	81:	nMoverToCorrect := nMoverToCorrect +1;
		IF nMoverToCorrect <= g_nMoverCount THEN
			fMoverOrientationRead    := ipMoverApplication[nMoverToCorrect].std.P_ActPosition.c; 
			fMoverOrientationCorrect := fMoverOrientationRead;
			 bDoRotationCorrection := FALSE;
			nStatePreparation := nStatePreparation + 1;	
		ELSE
			bDerterminedMoverOrientation := TRUE;
			nStatePreparation := nStatePreparation + 9;	
		END_IF
		
	82:	IF fMoverOrientationCorrect >= 0 THEN
			IF fMoverOrientationCorrect > 360.0 THEN
				fMoverOrientationCorrect := fMoverOrientationCorrect - 180.0;
				bDoRotationCorrection := TRUE;
			ELSE
				nStatePreparation := nStatePreparation + 1;
			END_IF
		ELSE
			IF fMoverOrientationCorrect < 360.0 THEN
				fMoverOrientationCorrect := fMoverOrientationCorrect + 180.0;
				bDoRotationCorrection := TRUE;
			ELSE
				nStatePreparation := nStatePreparation + 1;
			END_IF
		END_IF			
		
		
	83:	IF bDoRotationCorrection THEN
			
			fPosX := ipMoverApplication[nMoverToCorrect].std.P_ActPosition.x;
			fPosY := ipMoverApplication[nMoverToCorrect].std.P_ActPosition.y;
			fPosC := ipMoverApplication[nMoverToCorrect].std.P_ActPosition.c;
	
			CorrectionPos.SetValuesXYC(fPosX, fPosY, fMoverOrientationCorrect);	
	
			ipMoverApplication[nMoverToCorrect].std.SetMoverPosition('Correction', CorrectionPos);
			
			nStatePreparation := nStatePreparation + 1;	
		ELSE
			nStatePreparation := nStatePreparation - 2;
		END_IF
		
	84:
		IF ipMoverApplication[nMoverToCorrect].std.P_SetMoverPosition.Done THEN
			nStatePreparation := nStatePreparation - 3;
		ELSIF ipMoverApplication[nMoverToCorrect].std.P_SetMoverPosition.Error THEN
			nErrorID := ipMoverApplication[nMoverToCorrect].std.P_SetMoverPosition.ErrorID;
			ipVisuMessage.SetErrorMessage('Rotation-Angle modulo adaption', 'MoverPreparation', nStatePreparation, nErrorID);		
		END_IF
		

	90: nStatePreparation := 500;
	
			
	500: // Done
		nStatePreparation := 0;
		MoverPreparation := TRUE;		
			
		
	END_CASE


	ipVisuMessage.StateUpdate(nStatePreparation, 'MoverPreparation');
END_METHOD

METHOD MoverRecovery : BOOL
VAR_INPUT
	bReset	: BOOL;
END_VAR



VAR_INST

	// Dynamic limitations
	fVeloRec           				: LREAL := 250.0;
	fAccelRec    					: LREAL := 3000.0;
	fJerkRec            			: LREAL := 30000.0;
	
	fVeloTurn           			: LREAL :=  1800.0;
	fAccelTurn    					: LREAL :=   720.0;
	fJerkTurn            			: LREAL := 14400.0;		
	

	idx								: UDINT;	
	nTestCounter					: UDINT;
	nStateMoverRecovery				: INT;	
	bAllMoversDone					: BOOL;
	nForCounter						: UDINT;
	bStillBusy						: BOOL;
	nInitPositionToMoveTo			: UDINT;
	bAllMoversAtInitPosition		: BOOL;
	nInitPositionIndex	  			: UDINT;
	nMoverIndex			  			: UDINT;
	nMoversToInitPositionFound		: UDINT;
	nMoverToJoinTrack				: UDINT;
	nMoverToInitPosition			: UDINT;
	bTryMoveX						: BOOL;
	bTryMoveY						: BOOL;
	nCounterMoverToMove				: INT;	
	
	fInitialMoverPosition			: ARRAY [1..gc_nMaxNumberMovers,1..2] OF LREAL;
	bMoverSortedAlready				: ARRAY [1..gc_nMaxNumberMovers] OF BOOL;
	bMoverSkipInitPosition			: ARRAY [1..gc_nMaxNumberMovers] OF BOOL;
	bMoverToInitPosition			: ARRAY [1..gc_nMaxNumberMovers] OF BOOL;
	bMoverAtInitPosition			: ARRAY [1..gc_nMaxNumberMovers] OF BOOL;
	bMoverBlockedByMove				: ARRAY [1..gc_nMaxNumberMovers] OF BOOL;
	bInitPositionBlockedByMove		: ARRAY [1..gc_nMaxNumberMovers] OF BOOL;	
	bInitialMoverPositionDone		: ARRAY [1..gc_nMaxNumberMovers] OF BOOL;
	nMoverOnTheWayToInitPosition	: ARRAY [1..gc_nMaxNumberMovers] OF UDINT;
	fMoverDistanceToInitialPosition	: ARRAY [1..gc_nMaxNumberMovers] OF LREAL;
	fShortestDistance				: ARRAY [1..gc_nMaxNumberMovers] OF LREAL;
	nClosestMoverToInitPosition		: ARRAY [1..gc_nMaxNumberMovers] OF UDINT;
	nInitPositionMoverTable			: ARRAY [1..gc_nMaxNumberMovers] OF UDINT;
	nMoverRecoveryPosition			: ARRAY [1..gc_nMaxNumberMovers] OF UDINT;
	nJoinTrack						: ARRAY [1..gc_nMaxNumberMovers] OF UDINT;	
	
	fRotationMoverPosition			: ARRAY [1..gc_nMaxNumberMovers,1..2] OF LREAL;
	nMoverToRotationPosition		: UDINT;
	nRotationPositionToMoveTo		: UDINT;
	nMoverBackToInitPosition		: UDINT;

	sInfoText						: STRING;
	targetPos            	 		: PositionXYC;
    currentPos			     		: PositionXYC;
	nCmdReturnError					: UDINT;
	
	
//-----------------first Track run

	fTrackLengthTrack1  	: LREAL;
	fTrackLengthTrack2  	: LREAL;	
	fTrackLengthTrack3  	: LREAL;	
	
	bInitRunFlag			: BOOL;
	bInitRunDone			: BOOL;
	bOneMoverMoving			: BOOL;
	bAllMoversStandingStill	: BOOL;
	bMoversQueuing			: BOOL;
	
	TimerWaitForMovement	: TON;	
	
	
	nState 					: INT;	
	nStateInit				: INT;
	
	
	fbInitList				: FB_List;

	fPositionOnTrack			: LREAL;
	nStationIndex				: UINT;
	nNextStationTrackIndex 		: UINT;
	fNextStationWaitingPosition	: LREAL;
	nTrackIndex					: UDINT;
	nNextStationIndex			: UDINT;
	nListIdentifier				: UDINT;
	bFirstMoverIn				: BOOL;
	ClearTrig					: R_TRIG;
	fMoverPosition				: LREAL;
	fMoverVelocity				: LREAL;
	fMoverAcceleration			: LREAL;
	fMoverJerk					: LREAL;
	strInfo						: STRING;
	
	fMoverSpace					: LREAL;
	fWaitingPositionStation01	: LREAL;
	fWaitingPositionStation02	: LREAL;	
	fWaitingPositionStation03	: LREAL;	
	fWaitingPositionStation04	: LREAL;	
	fWaitingPositionStation05b	: LREAL;	
	fWaitingPositionStation05c	: LREAL;
	
	stMoveParameters 	: ST_MoveOnTrackOptions; 
	strInfoHistory		: ARRAY[0..10] OF STRING;
	
	nResult				: DINT;
	sMessage			: STRING;
	
	
	stJoinTrackOptions		: ST_JoinTrackOptions;
	stMoveOptionsCurve		: ST_MoveCOptions;	

	
	
	nMoverToTurnBack				: UDINT;
	fRecoveryRotTarget				: LREAL;
	fRecoveryRotVel					: LREAL :=  360.0;
	fRecoveryRotAcc					: LREAL := 1800.0;
	fRecoveryRotJerk				: LREAL := 9000.0;
	stRotationOptions				: ST_MoveCOptions;
	
	
	LeavOptions	: ST_LeaveTrackOptions;
	
END_VAR


VAR_INST
	nMoverToTurn					: UDINT;

	fbMoverTarget		: FB_MoverTarget;
	nErrorCode			: DINT;
	bError				: BOOL;
	sInfoMessage		: STRING;

	
END_VAR
IF bReset THEN
	nStateMoverRecovery := 0;
	MoverRecovery := TRUE;
END_IF



CASE nStateMoverRecovery OF

	0:	// Starting mover recovery
		nStateMoverRecovery := 50;
			
	(***************************************************************************************)
	(* Mover Recovery Part1: Checking for unfinished rotation                              *)
	(***************************************************************************************)     			
		
	50:		// Turn rotation angle to closets quarter-angle 
			ipVisuMessage.SetInfoMessage('Clearing rotation', 'Recovery', nStateMoverRecovery);

			nMoverToTurn := 0;
			nStateMoverRecovery := nStateMoverRecovery +1;
			
	51:  	nMoverToTurn := nMoverToTurn +1;
			IF nMoverToTurn > g_nMoverCount THEN
				nStateMoverRecovery := nStateMoverRecovery +3;
			ELSE
				IF ipMoverApplication[nMoverToTurn].std.P_IsPresent THEN

					fRecoveryRotTarget 				  := ipMoverApplication[nMoverToTurn].std.P_ClosestQuaterAngle;	
					stRotationOptions.additionalTurns := 0;
					stRotationOptions.direction		  := Tc3_Mc3PlanarMotion.MC_direction.mcDirectionNonModulo;	
					
					ipMoverApplication[nMoverToTurn].std.MoveC('Recovery - unfinished rotation', fRecoveryRotTarget, fRecoveryRotVel, fRecoveryRotAcc, fRecoveryRotAcc, fRecoveryRotJerk, stRotationOptions);
					nStateMoverRecovery := nStateMoverRecovery +1;				
				END_IF	
			END_IF

	52:		IF ipMoverApplication[nMoverToTurn].std.P_MoveC.Done THEN
				nStateMoverRecovery := nStateMoverRecovery -1;	
			ELSIF ipMoverApplication[nMoverToTurn].std.P_MoveC.Error THEN
				nStateMoverRecovery := nStateMoverRecovery +1;	
			END_IF
 
	53:		// Check error ID and react accordingly
			nErrorID := ipMoverApplication[nMoverToTurn].std.P_MoveC.ErrorID;	
			
			// In case rotation is not possible due to collision with another mover proceed without rotation correction.
			IF nErrorID = 33158 THEN
				nStateMoverRecovery := nStateMoverRecovery -2;	
			END_IF
						
	54:		nStateMoverRecovery := 100;		
			
			
	(*******************************************************************************************)
	(* Mover Recovery Part2: Separating all movers and move each of them to a corner position. *)
	(*******************************************************************************************)    			
		
	100: 
		ipVisuMessage.SetInfoMessage('Separating all movers', 'Recovery', nStateMoverRecovery);
		IF fbMoverTarget.Clear() THEN
			nStateMoverRecovery := nStateMoverRecovery +10;
		END_IF
	
	110:
		bError := FALSE;
		FOR idx:=1 TO g_nMoverCount DO
			IF ipMoverApplication[idx].std.P_IsPresent THEN
				fbMoverTarget.AddMover(ipMoverApplication[idx]);
				IF fbMoverTarget.P_ErrorWarningCode < 0 THEN
					bError := TRUE;
				END_IF
			END_IF
		END_FOR
		
		IF bError THEN
			sInfoMessage := fbMoverTarget.P_Info;
		ELSE
			nStateMoverRecovery := nStateMoverRecovery +10;
		END_IF
			
	120:
		fbMoverTarget.AddPosition(120.0, 120.0);
		fbMoverTarget.AddPosition(120.0, 600.0);
		fbMoverTarget.AddPosition(840.0, 600.0);
		fbMoverTarget.AddPosition(840.0, 120.0);
		
		fbMoverTarget.SetDynamics(250.0, 1000.0, 10000.0);
		
		IF fbMoverTarget.P_ErrorWarningCode < 0 THEN
			sInfoMessage := fbMoverTarget.P_Info;
		ELSE
			nStateMoverRecovery := nStateMoverRecovery +10;
		END_IF
		

	130:
		  sMessage := fbMoverTarget.P_Info;
		nErrorCode := fbMoverTarget.P_ErrorWarningCode;	

		IF fbMoverTarget.MoversToTarget() THEN
			nStateMoverRecovery := 300;
		END_IF
					
	
	(***************************************************************************************)
	(* Mover Recovery Part3: All movers join the outer-track							   *)
	(***************************************************************************************)  	
					
			
	300:	// All movers go on track
			ipVisuMessage.SetInfoMessage('All movers join track', 'Recovery', nStateMoverRecovery);
	
			FOR nForCounter := 1 TO g_nMoverCount DO
				IF ipMoverApplication[nForCounter].std.P_SetPosition.x > 480.0 THEN
					nJoinTrack[nForCounter] := 3;	
				ELSE
					nJoinTrack[nForCounter] := 1;	
				END_IF
			END_FOR
			nStateMoverRecovery := nStateMoverRecovery +1;	
				
	301:	IF nMoverToJoinTrack < g_nMoverCount THEN
				nMoverToJoinTrack := nMoverToJoinTrack +1;
				nStateMoverRecovery := nStateMoverRecovery +1;
			ELSE
				nMoverToJoinTrack := 0;
				nStateMoverRecovery := nStateMoverRecovery + 2; 
			END_IF
				
	302:	stJoinTrackOptions.useOrientation := FALSE;
	
			sInfoText := 'Recovery, join TrackID: ';
			sInfoText := CONCAT(sInfoText, UDINT_TO_STRING(nJoinTrack[nMoverToJoinTrack]));
			
			IF ipMoverApplication[nMoverToJoinTrack].std.JoinTrack( sInfoText,
																	ipTrack[nJoinTrack[nMoverToJoinTrack]].std,
																    fVeloRec,
																	fAccelRec,
																	fJerkRec,
																	stJoinTrackOptions )
			THEN
				ipMoverApplication[nMoverToJoinTrack].P_TrackId := nJoinTrack[nMoverToJoinTrack];
				nStateMoverRecovery := nStateMoverRecovery -1;
			END_IF
			
				
			
			
	303:	bDone := TRUE;
			FOR nForCounter := 1 TO g_nMoverCount DO
				bDone := bDone AND ipMoverApplication[nForCounter].std.P_JoinTrack.Done;
			END_FOR
			
			IF bDone THEN
				nStateMoverRecovery := nStateMoverRecovery + 7;
			END_IF
		
	310:  // Wait for all movers on-track
			bDone := TRUE;
			FOR nForCounter := 1 TO g_nMoverCount DO
				bDone := bDone AND ipMoverApplication[nForCounter].std.P_JoinTrack.Done;
			END_FOR
			IF bDone THEN
				nStateMoverRecovery := 400;
			END_IF
	
				
	(***************************************************************************************)
	(* Mover Recovery Part4: Adding all movers to the Initialization-List and sort them    *)
	(*                       ascending.                              				       *)
	(***************************************************************************************)  			
				
	400:	ipVisuMessage.SetInfoMessage('Sorting all movers', 'Recovery', nStateMoverRecovery);
			IF fbInitList.ClearList() THEN
				nStateMoverRecovery := nStateMoverRecovery + 1;
			END_IF
			
	401:	IF fbInitList.ClearTrackOrder() THEN
				nStateMoverRecovery := nStateMoverRecovery + 9;
			END_IF
	
			
	410:	// Adding all movers to the Initialization-List
			FOR nForCounter := 1 TO g_nMoverCount DO
				fbInitList.AddMover(ipMoverApplication[nForCounter].std);
			END_FOR				
			nStateMoverRecovery := nStateMoverRecovery + 10;
			
			
	420: 	// Adding Track-Order to the Initialization-List for Sorting-Order
			IF fbInitList.AddTrack(ipTrack[1].std) > 0 THEN
				nStateMoverRecovery := nStateMoverRecovery + 1;
			ELSE
				 nResult := fbInitList.P_nResult;
				sMessage := fbInitList.P_sMessage;	
			END_IF
			
	421: 	IF fbInitList.AddTrack(ipTrack[3].std) > 0 THEN
				nStateMoverRecovery := nStateMoverRecovery + 1;
			ELSE
				 nResult := fbInitList.P_nResult;
				sMessage := fbInitList.P_sMessage;	
			END_IF			
						
 	422:	nStateMoverRecovery := 450;
				
	450:	// Sorting all movers 
			fbInitList.P_SortingDirection := eSortingDirection.ascending;
			fbInitList.P_SortingOrigin := 0.0;
	
			 nResult := fbInitList.SortList();
			sMessage := fbInitList.P_sMessage;
			
			IF nResult > 0 THEN
				// Sorting succesful - will return the number of movers sorted e.g. 4
				nStateMoverRecovery:= nStateMoverRecovery + 10;
			ELSIF nResult = 0 THEN
				;// Sorting 
			ELSIF nResult < 0 THEN
				// sorting Error - Check error code and error message
				nStateMoverRecovery:= nStateMoverRecovery +1;
			END_IF
			
	451:	// Check error message and act accordingly		
			 nResult := fbInitList.P_nResult;
			sMessage := fbInitList.P_sMessage;				
	
			
	460:	nStateMoverRecovery:= 500;			
	

	
	(***************************************************************************************)
	(* Mover Recovery Part5: Initialization-Run                                            *)
	(*						 - Sending/Adding each mover to its next closest station       *)
	(*						 - From there on each station takes care of the init-run       *)
	(* 						 - Movers will queu in in front of station 01 				   *)
	(***************************************************************************************)  

	500: // Init all variables 
		ipVisuMessage.SetInfoMessage('Mover init-run', 'Recovery', nStateMoverRecovery);
	
					bOneMoverMoving := FALSE;
			bAllMoversStandingStill := FALSE;
					   bInitRunDone := FALSE;
	
				   nStateMoverRecovery := nStateMoverRecovery + 10;
	
	510: // Check for next Mover
		IF fbInitList.P_FirstInList <> 0 THEN
				 nMoverIndex := fbInitList.P_FirstInList.P_Id;
				 nTrackIndex := ipMoverApplication[nMoverIndex].P_TrackId;
			fPositionOnTrack := ipMoverApplication[nMoverIndex].std.P_SetOnTrack.SetPos;
			
			      bFirstMoverIn := TRUE;
			nStateMoverRecovery := nStateMoverRecovery + 10;
		ELSE
			IF bFirstMoverIn THEN
				nStateMoverRecovery := 600;
			ELSE
				// Init-Run completed
				bInitRunFlag := FALSE;
				nStateMoverRecovery := 1000;	
			END_IF
		END_IF
			
		
	520: // Figuring out the next station the mover has to travel to:
		fMoverSpace := 155.0 + 5.0;
	
		fWaitingPositionStation01	:= ipTrack[1].P_TrackLength/2.0 - fMoverSpace;	
		fWaitingPositionStation02	:= ipTrack[2].P_TrackLength/2.0 - fMoverSpace;	
		fWaitingPositionStation03	:= ipTrack[3].P_TrackLength/2.0 - fMoverSpace;
		fWaitingPositionStation04	:= ipTrack[1].P_TrackLength - fMoverSpace;	
		fWaitingPositionStation05b	:= ipTrack[3].P_TrackLength - fMoverSpace;	
		fWaitingPositionStation05c	:= ipTrack[2].P_TrackLength - fMoverSpace;	
	
		nListIdentifier := 0;
		CASE nTrackIndex OF		
		1:	// Mover on Track01 / Station01
			IF fPositionOnTrack <= fWaitingPositionStation01 THEN
				nNextStationIndex := 1;
				  nListIdentifier := 11;
			ELSE
				nNextStationIndex := 4;
				  nListIdentifier := 14;
			END_IF	
	
		2:	// Mover on Track02 / Station02
			IF fPositionOnTrack <= fWaitingPositionStation02 THEN
				nNextStationIndex := 2;
				  nListIdentifier := 22;
			ELSE
				nNextStationIndex := 5;
				  nListIdentifier := 25;
			END_IF			
		
		3:	// Mover on Track03 / Station 03
			IF fPositionOnTrack <= fWaitingPositionStation03 THEN
				nNextStationIndex := 3;
				  nListIdentifier := 33;
			ELSE
				nNextStationIndex := 5;
				  nListIdentifier := 35;
			END_IF			
		END_CASE
		
		nStateMoverRecovery := nStateMoverRecovery + 10;
			
			
	530: // Calculating the position the mover has to move to next:
		nNextStationTrackIndex := 0;
		
		CASE nNextStationIndex OF
			1:	nNextStationTrackIndex      := 1;
				fNextStationWaitingPosition	:= fWaitingPositionStation01;	
			
			2:	nNextStationTrackIndex      := 2;
				fNextStationWaitingPosition	:= fWaitingPositionStation02;			
			
			3:	nNextStationTrackIndex      := 3;
				fNextStationWaitingPosition	:= fWaitingPositionStation01;			
			
			4:	nNextStationTrackIndex      := 1;
				fNextStationWaitingPosition	:= fWaitingPositionStation04;				
				
			5:	IF nTrackIndex = 2 THEN
					nNextStationTrackIndex := 2;
					fNextStationWaitingPosition	:= fWaitingPositionStation05c;	
				ELSIF nTrackIndex = 3 THEN
					nNextStationTrackIndex := 3;
					fNextStationWaitingPosition	:= fWaitingPositionStation05b;	
				END_IF									
		END_CASE
			
		IF nNextStationTrackIndex > 0 THEN
			nStateMoverRecovery := nStateMoverRecovery + 10;
		END_IF
	
	
	540: 	// Send mover to the next station
			fMoverPosition     := fNextStationWaitingPosition;
			fMoverVelocity     :=    300.0;
			fMoverAcceleration :=  1_000.0;
			fMoverJerk         := 10_000.0;	
	
			stMoveParameters.direction := Tc3_Mc3PlanarMotion.MC_DIRECTION.mcDirectionPositive;
			stMoveParameters.gap       := 240.0;
			
			strInfo := 'Recovery: ';
			strInfo := CONCAT(strInfo, ' Mover: ');
			strInfo := CONCAT(strInfo, UDINT_TO_STRING(nMoverIndex));
			strInfo := CONCAT(strInfo, ' move to Station:' );
			strInfo := CONCAT(strInfo, UDINT_TO_STRING(nNextStationIndex));
			
		
			IF NOT ipMoverApplication[nMoverIndex].std.P_MoveOnTrack.Busy THEN
	
				FOR idx:=10 TO 1 BY -1 DO 
					strInfoHistory[idx] := strInfoHistory[idx-1];
				END_FOR
				strInfoHistory[0] := strInfo;		
			
				ipMoverApplication[nMoverIndex].std.MoveOnTrack( strInfo,
																 ipTrack[nNextStationTrackIndex].std,
																 fMoverPosition,
																 fMoverVelocity,
																 fMoverAcceleration,
																 fMoverJerk,
																 stMoveParameters.gap,
																 stMoveParameters.direction);
				nStateMoverRecovery := nStateMoverRecovery +1;
				
				
				ipMoverApplication[nMoverIndex].P_ProductData.bInitRun            := TRUE;
				ipMoverApplication[nMoverIndex].P_ProductData.nDestinationProcess := 0;
			END_IF	
			
	541: 
		IF ipMoverApplication[nMoverIndex].std.P_MoveOnTrack.Active THEN
			nStateMoverRecovery := nStateMoverRecovery + 9;
		END_IF
			
	 
	550: // Mover to the list of the next station
		CASE nListIdentifier OF
		11:	ipStation[1].P_List_Station.AddMover(fbInitList.RemoveFirstInList());
		14: ipStation[4].P_List_Switch_Input_A.AddMover(fbInitList.RemoveFirstInList());
		
		22: ipStation[2].P_List_Station.AddMover(fbInitList.RemoveFirstInList());
		25:	ipStation[5].P_List_Switch_Input_C.AddMover(fbInitList.RemoveFirstInList());
		
		33: ipStation[3].P_List_Station.AddMover(fbInitList.RemoveFirstInList());
		35: ipStation[5].P_List_Switch_Input_B.AddMover(fbInitList.RemoveFirstInList());
		END_CASE
	
		IF nListIdentifier > 0 THEN
			nStateMoverRecovery := 510;	
		END_IF
		

	600: // Set all stations into "Init-Run" Mode	
		FOR idx:=1 TO gc_NumberStations DO
			ipStation[idx].P_eProcessMode := E_ProcessMode.InitRun;
		END_FOR	
		nStateMoverRecovery := nStateMoverRecovery + 10;	
		
		
	610: // Wait till at least one mover started moving, or timeout if no movement at all.	
		bOneMoverMoving := FALSE;
		FOR idx:=1 TO g_nMoverCount DO	
			IF ABS(ipMoverApplication[idx].std.P_SetVelocity.x) > 0.1
			OR ABS(ipMoverApplication[idx].std.P_SetVelocity.y) > 0.1
			THEN
				bOneMoverMoving := TRUE;
			END_IF
		END_FOR		
	
		TimerWaitForMovement(IN:=TRUE, PT:=T#2S);
		
		IF bOneMoverMoving 
		OR TimerWaitForMovement.Q 
		THEN
			TimerWaitForMovement(IN:=FALSE);
			nStateMoverRecovery := nStateMoverRecovery + 10;			
		END_IF
		
	
	620: // Wait till all movers are standing still	
		bAllMoversStandingStill := TRUE;
		FOR idx:=1 TO g_nMoverCount DO			
			IF ipMoverApplication[idx].std.P_IsMovingXY THEN
				bAllMoversStandingStill := FALSE;
			END_IF
		END_FOR
		
		IF bAllMoversStandingStill THEN
			nStateMoverRecovery := nStateMoverRecovery + 10;				
		END_IF
		
		
	630: // Init-Run done
		FOR idx:=1 TO gc_NumberStations DO
			ipStation[idx].P_eProcessMode := E_ProcessMode.None;
		END_FOR		

			   bInitRunDone := TRUE;
		nStateMoverRecovery := 1000;		
			
	
	1000:// Mover recovery done
		ipVisuMessage.SetInfoMessage('Mover recovery done', 'Recovery', nStateMoverRecovery);
	
			   MoverRecovery := TRUE;
		 nStateMoverRecovery := 0;	
			

END_CASE


ipVisuMessage.StateUpdate(nStateMoverRecovery, 'Recovery');
END_METHOD

PROPERTY P_AbortingSequence : DINT
GET
P_AbortingSequence := nAbortingSequence;
END_GET
END_PROPERTY

PROPERTY P_Alarm : ST_VisuMessage
GET
END_GET
END_PROPERTY

PROPERTY P_ExecutingSequence : DINT
GET
P_ExecutingSequence := nExecutingSequence;
END_GET
END_PROPERTY

PROPERTY P_MoverError : BOOL
GET
P_MoverError := bMoverError;
END_GET
SET
bMoverError := P_MoverError;
END_SET
END_PROPERTY

PROPERTY PUBLIC P_ResettingSequence : DINT
GET
P_ResettingSequence := nResettingSequence;
END_GET
END_PROPERTY

PROPERTY PUBLIC P_StartingSequence : DINT
GET
P_StartingSequence := nPrepareSequence;
END_GET
END_PROPERTY

PROPERTY PUBLIC P_StartupSequence : DINT
GET
P_StartupSequence := nStartupSequence;
END_GET
END_PROPERTY

METHOD Prepare : BOOL


VAR_INST
	Test : LREAL;	

	bAllMoversDone				: BOOL; 	
	
	nStationToInit				: UINT;
	

	nMoversFound				: UDINT;
	
	sTextTemp					: STRING;
	

	
	nTestCounter				: UDINT;
	
	
	
END_VAR
nErrorID := 0;

CASE nPrepareSequence OF 
	

	0:	// Enter
		nPrepareSequence := 10;	

	
	(***************************************************************************************)
	(* Starting Part 1: Getting everything ready...                                        *)
	(***************************************************************************************) 		
			
	10: // EnableGroup
		IF ipMotionSystem.EnableGroup() THEN
			ipVisuMessage.SetInfoMessage('ENABLE Group', 'Prepare', nPrepareSequence);
			nPrepareSequence := nPrepareSequence + 1;
		END_IF
		
	11: IF ipMotionSystem.P_EnableGroup.Done THEN
			nPrepareSequence := nPrepareSequence +9;
		ELSIF ipMotionSystem.P_EnableGroup.Error THEN
			nPrepareSequence := nPrepareSequence + 1;
		END_IF	
			
	12:	// Check error ID and react accordingly
		nErrorID := ipMotionSystem.P_EnableGroup.ErrorID;
		ipVisuMessage.SetErrorMessage('ENABLE Group failed', 'Prepare', nPrepareSequence, nErrorID);		
		
		
	20: // Adding Environment to Group
		IF ipMotionSystem.AddEnvironmentToGroup() THEN
			ipVisuMessage.SetInfoMessage('Add Group to Environment', 'Prepare', nPrepareSequence);
			nPrepareSequence := nPrepareSequence +1;
		END_IF	
		
	21: IF ipMotionSystem.P_AddEnviromentToGroup.Done THEN
			nPrepareSequence := nPrepareSequence +9;
		ELSIF ipMotionSystem.P_AddEnviromentToGroup.Error THEN
			nPrepareSequence := nPrepareSequence +1;		
		END_IF	
		
	22:	// Check error ID and react accordingly
		nErrorID := ipMotionSystem.P_AddEnviromentToGroup.ErrorID;
		ipVisuMessage.SetErrorMessage('Add Group to Environment failed', 'Prepare', nPrepareSequence, nErrorID);			
				
				
	30: // Enable all tracks
		IF ipMotionSystem.EnableTracks() THEN
			ipVisuMessage.SetInfoMessage('ENABLE Tracks', 'Prepare', nPrepareSequence);
			nPrepareSequence := nPrepareSequence +1;
		END_IF
		
	31:	
		IF ipMotionSystem.P_EnableTracks.Done THEN
			nPrepareSequence := nPrepareSequence +9;
		ELSIF ipMotionSystem.P_EnableTracks.Error THEN
			nPrepareSequence := nPrepareSequence +1;		
		END_IF
		
	32:	// Check error ID and react accordingly
		nErrorID := ipMotionSystem.P_EnableTracks.ErrorID;
		ipVisuMessage.SetErrorMessage('ENABLE Tracks failed', 'Prepare', nPrepareSequence, nErrorID);				
		
			
	40: // Adding all tracks to the group
		IF ipMotionSystem.AddTracksToGroup() THEN
			ipVisuMessage.SetInfoMessage('Add tracks to Group', 'Prepare', nPrepareSequence);
			nPrepareSequence := nPrepareSequence +1;
		END_IF
	
	41: IF ipMotionSystem.P_AddTracksToGroup.Done THEN
			nPrepareSequence := nPrepareSequence +9;
		ELSIF ipMotionSystem.P_AddTracksToGroup.Error THEN
			nPrepareSequence := nPrepareSequence +1;
		END_IF
		
	42:	// Check error ID and react accordingly120
		nErrorID := ipMotionSystem.P_AddTracksToGroup.ErrorID;
		ipVisuMessage.SetErrorMessage('Add tracks to Group failed', 'Prepare', nPrepareSequence, nErrorID);				

	
	50: // Init all stations
		nStationToInit := 0;
		nPrepareSequence := nPrepareSequence +1;

	51:	nStationToInit := nStationToInit +1;
		IF nStationToInit <= gc_NumberStations THEN
			ipVisuMessage.SetInfoMessage(CONCAT('Init Station:' ,UINT_TO_STRING(nStationToInit)), 'Prepare', nPrepareSequence);
			nPrepareSequence := nPrepareSequence +1;
		ELSE
			nPrepareSequence := nPrepareSequence +9;
		END_IF	
				
	52: IF ipStation[nStationToInit].Init() THEN
			nPrepareSequence := nPrepareSequence -1;
		END_IF

		
	60:	nPrepareSequence := 100;
	
	
	
	100: // Prepare all movers
		IF MoverPreparation(bReset:=TRUE) THEN
			nPrepareSequence := nPrepareSequence + 1;
		END_IF
		
	101:
		IF MoverPreparation(bReset:=FALSE) THEN
			nPrepareSequence := nPrepareSequence + 9;
		END_IF	
		
		
		
	110: nPrepareSequence := 160;
		
	
	160:// Enable all movers
		IF ipMotionSystem.EnableMovers() THEN
			ipVisuMessage.SetInfoMessage('ENABLE all movers', 'Prepare', nPrepareSequence);
			nPrepareSequence := nPrepareSequence + 1;
		END_IF
	
	161: 
		IF ipMotionSystem.P_EnableMovers.Done THEN
			nPrepareSequence := nPrepareSequence +9;
		ELSIF ipMotionSystem.P_EnableMovers.Error THEN

			nPrepareSequence := nPrepareSequence + 1;
		END_IF	
			
	162:// Error = Not able to enable movers e.g. mover was not able to reach it's flight hight due to high payload 
		nErrorID := ipMotionSystem.P_EnableMovers.ErrorID;	
		ipVisuMessage.SetErrorMessage('ENABLE all movers failed', 'Prepare', nPrepareSequence, nErrorID);	
	

		
	
    170: // Adding movers to the group
		IF ipMotionSystem.AddMoversToGroup() THEN
			ipVisuMessage.SetInfoMessage('Add movers to Group', 'Prepare', nPrepareSequence);
			nPrepareSequence := nPrepareSequence + 1;
		END_IF
	
    171: IF ipMotionSystem.P_AddMoversToGroup.Done THEN
			nPrepareSequence := nPrepareSequence +9;
		ELSIF ipMotionSystem.P_AddMoversToGroup.Error THEN
			nPrepareSequence := nPrepareSequence + 1;
		END_IF	
	
    172:// Check error ID and react accordingly
		nErrorID := ipMotionSystem.P_AddMoversToGroup.ErrorID;
		ipVisuMessage.SetErrorMessage('Add movers to Group failed', 'Prepare', nPrepareSequence, nErrorID);	
	
	
	180: nPrepareSequence := 200;			
				

	(***************************************************************************************)
	(* Starting Part 3: Organize all movers to get ready for the machine process           *)
	(***************************************************************************************) 		
			
	200:  // Mover Recovery/Sorting
		IF MoverRecovery(bReset:=TRUE) THEN;
			nPrepareSequence := nPrepareSequence +1;	
		END_IF	
	
	201:
		IF MoverRecovery(bReset:=FALSE) THEN
			nPrepareSequence := nPrepareSequence +9;		
		END_IF
	
			
	210:  // Prepare sequence done
		ipVisuMessage.SetInfoMessage('PREPARE finished', 'Prepare', 0);
					 Prepare := TRUE;			 
			nPrepareSequence := 0; 
			
		
END_CASE


ipVisuMessage.StateUpdate(nPrepareSequence, 'Prepare');
END_METHOD

METHOD Reset : BOOL
VAR_INPUT
END_VAR
	
	// Resetting all necesarry internal data 
	bMoverError := FALSE;



	Reset := TRUE;
END_METHOD

METHOD Resetting : BOOL
VAR_INPUT
END_VAR




VAR_INST
	
	nTrackToEnable		: UDINT;
	stProductDataClear 	: ST_ProductData;
	
END_VAR
nErrorID := 0;

CASE nResettingSequence OF 
	
	0: // Enter 
		nResettingSequence := 10;
		
		
		
	10: // Reset all movers
		IF ipMotionSystem.ResetMovers() THEN
			ipVisuMessage.SetInfoMessage('RESET all movers', 'Resetting', nResettingSequence);
			nResettingSequence := nResettingSequence +1;			
		END_IF
		
	11: IF ipMotionSystem.P_ResetMovers.Done THEN
			nResettingSequence := nResettingSequence +9;
		ELSIF ipMotionSystem.P_ResetMovers.Error THEN
			nResettingSequence := nResettingSequence +1;	
		END_IF

	12:	// Check error ID and react accordingly
		nErrorID := ipMotionSystem.P_EnableMovers.ErrorID;
		ipVisuMessage.SetErrorMessage('RESET movers failed', 'Resetting', nResettingSequence, nErrorID);					
		
		
		
	20:	// Reset all tracks
		IF ipMotionSystem.ResetTracks() THEN
			ipVisuMessage.SetInfoMessage('RESET all tracks', 'Resetting', nResettingSequence);
			nResettingSequence := nResettingSequence +1;
		END_IF
		
	21: IF ipMotionSystem.P_ResetTracks.Done THEN
			nResettingSequence := nResettingSequence +9;
	 	ELSIF ipMotionSystem.P_ResetTracks.Error THEN
			nResettingSequence := nResettingSequence +1;	
		END_IF
	
	22:	// Check error ID and react accordingly
		nErrorID := ipMotionSystem.P_EnableMovers.ErrorID;
		ipVisuMessage.SetErrorMessage('RESET tracks failed', 'Resetting', nResettingSequence, nErrorID);			
		
	
		
	30:	// Reset MotionSystemApplication
		IF ipMotionSystemApplication.Reset() THEN
			ipVisuMessage.SetInfoMessage('RESET MotionSystemApplication', 'Resetting', nResettingSequence);
			nResettingSequence := nResettingSequence +10;
		END_IF
	
				
	40:  // Cleaning all process data
		FOR idx:=1 TO g_nMoverCount DO
			ipMoverApplication[idx].P_ProductData := stProductDataClear;
		END_FOR
		nResettingSequence := 100;
		
	
	100: // Reset done
		ipVisuMessage.SetInfoMessage('RESET finished', 'Resetting', 0);
	
		nResettingSequence := 0; 
		         Resetting := TRUE;

END_CASE



ipVisuMessage.StateUpdate(nResettingSequence, 'Resetting');
END_METHOD

METHOD Startup : BOOL
VAR
	aMoverDetectionSetup	: ARRAY[1..3] OF ST_TcIoMoverDetectionSetup;
END_VAR

VAR_INST
	
	// Tracks
	nTrackToInit			: UDINT;
	nTrackToGroup			: UDINT;
	sErrorInfo				: STRING;
	
	stHaltDynamics			: ST_HaltDynamics;
	
END_VAR


CASE nStartupSequence OF 
	
	0: // Enter
		IF ipVisuMessage <> 0 THEN
			nStartupSequence := nStartupSequence +1;
		END_IF

 
	1: // Wait for initialization
		IF ipMotionSystem.P_SystemInitialized THEN
			ipVisuMessage.SetInfoMessage('MotionSystem initialized', 'Startup', nStartupSequence);	
			nStartupSequence := 10;
		ELSE
			ipVisuMessage.SetInfoMessage('Waiting for initialization of MotionSystem', 'Startup', nStartupSequence);	
		END_IF
	
	
	10: // Initialization of all tracks	
		    nTrackToInit := 0;
		nStartupSequence := nStartupSequence +1;
	
	11: // Track number count
		IF nTrackToInit < gc_NumberTracks THEN
			nTrackToInit := nTrackToInit + 1;
			nStartupSequence := nStartupSequence +1;
					
			sTextTemp := 'Initializing Track: ';
			sTextTemp := CONCAT(sTextTemp, UDINT_TO_STRING(nTrackToInit));			
			ipVisuMessage.SetInfoMessage(sTextTemp, 'Startup', nStartupSequence);
		ELSE
			    nTrackToInit := 0;
			nStartupSequence := 20;
		END_IF
				
	12:	// Clear track data
		IF ipTrack[nTrackToInit].Clear() THEN
			nStartupSequence := nStartupSequence +1;
		END_IF
		
	13: // Build the track
		IF ipTrack[nTrackToInit].Initialize(nTrackToInit) THEN	
			nStartupSequence := 11;
		ELSE
			IF ipTrack[nTrackToInit].P_Error THEN
				nStartupSequence := nStartupSequence +1;
			END_IF
		END_IF
		
	14:	// In case of error react accordingly
		sErrorInfo := ipTrack[nTrackToInit].P_ErrorInfo;
				
		sTextTemp := CONCAT(sErrorInfo, UDINT_TO_STRING(nTrackToInit));			
		ipVisuMessage.SetErrorMessage(sTextTemp, 'Startup', nStartupSequence, 0);
	
	
	20: // Setting halt-dynamics for all movers
		stHaltDynamics.Mode := E_HaltDynamicsMode.AxisX_AxisY_CoordinatedOnPath;
	
		stHaltDynamics.PathXY.fVelocity		:=    500.0;
		stHaltDynamics.PathXY.fAcceleration	:=  10000.0;
		stHaltDynamics.PathXY.fDeceleration	:=  10000.0;
		stHaltDynamics.PathXY.fJerk			:= 100000.0;

		stHaltDynamics.AxisX.fVelocity		:=    500.0;
		stHaltDynamics.AxisX.fAcceleration	:=  10000.0;
		stHaltDynamics.AxisX.fDeceleration	:=  10000.0;
		stHaltDynamics.AxisX.fJerk			:= 100000.0;

		stHaltDynamics.AxisY.fVelocity		:=    500.0;
		stHaltDynamics.AxisY.fAcceleration	:=  10000.0;
		stHaltDynamics.AxisY.fDeceleration	:=  10000.0;
		stHaltDynamics.AxisY.fJerk			:= 100000.0;

		stHaltDynamics.AxisZ.fVelocity		:=    500.0;
		stHaltDynamics.AxisZ.fAcceleration	:=  10000.0;
		stHaltDynamics.AxisZ.fDeceleration	:=  10000.0;
		stHaltDynamics.AxisZ.fJerk			:= 100000.0;		
		
		stHaltDynamics.AxisA.fVelocity		:=     10.0;
		stHaltDynamics.AxisA.fAcceleration	:=    100.0;
		stHaltDynamics.AxisA.fDeceleration	:=    100.0;	
		stHaltDynamics.AxisA.fJerk          :=    100.0;		
		
		stHaltDynamics.AxisB.fVelocity		:=     10.0;
		stHaltDynamics.AxisB.fAcceleration	:=    100.0;
		stHaltDynamics.AxisB.fDeceleration	:=    100.0;	
		stHaltDynamics.AxisB.fJerk          :=    100.0;			
		
		stHaltDynamics.AxisC.fVelocity		:=     36.0;
		stHaltDynamics.AxisC.fAcceleration	:=    360.0;
		stHaltDynamics.AxisC.fDeceleration	:=    360.0;	
		stHaltDynamics.AxisC.fJerk          :=    360.0;
		
		FOR idx:=1 TO g_nMoverCount DO
			ipMoverApplication[idx].std.P_HaltDynamics := stHaltDynamics;
		END_FOR
		
		nStartupSequence := 100;


	100: // Start-Up Done!
		ipVisuMessage.SetInfoMessage('START-UP finished', 'Startup', 0);				
		Startup := TRUE;
		
END_CASE


ipVisuMessage.StateUpdate(nStartupSequence, 'Startup');
END_METHOD

PROPERTY std : I_MotionSystem
GET
IF ipMotionSystem <> 0 THEN
	std := ipMotionSystem;	
END_IF
END_GET
SET
ipMotionSystem := std;
END_SET
END_PROPERTY

END_FUNCTION_BLOCK

// ---- 2_Application/Machine/FB_MoverTarget.TcPOU
FUNCTION_BLOCK FB_MoverTarget
VAR_INPUT
END_VAR
VAR_OUTPUT
END_VAR
VAR
	
	positionList		: ARRAY[1..gc_nMoverCountConfigured] OF ST_PositionXY;
	nPositionCount		: UDINT;
	moverList			: ARRAY[1..gc_nMoverCountConfigured] OF I_MoverApplication;	
	nMoversInList		: UDINT;
	
	nErrorWarningCode 	: DINT;
	sMessage 			: STRING;
	
	idx					: UDINT;
	
	recoverVelocity					: LREAL :=   250.0;
	recoveryAcceleration			: LREAL :=  1000.0;
	recoveryJerk					: LREAL := 10000.0;
	
	fShiftDistanceY			: LREAL;
	fShiftDistanceX			: LREAL;
	
	nStateMove						: DINT;
END_VAR

METHOD AddMover : BOOL
VAR_INPUT
	ipMover		: I_MoverApplication;
END_VAR



VAR
	bMoverInList	: BOOL;
END_VAR


	IF ipMover <> 0 THEN
	
		nMoversInList := 0;
		bMoverInList  := FALSE;
		FOR idx:=1 TO gc_nMoverCountConfigured DO
			IF moverList[idx] <> 0 THEN
				nMoversInList := nMoversInList +1;
				IF moverList[idx].std.P_Id = ipMover.std.P_Id THEN
					bMoverInList := TRUE;
				END_IF				
			END_IF
		END_FOR
		
		IF NOT bMoverInList THEN
			nMoversInList := nMoversInList +1;
			moverList[nMoversInList] := ipMover;
			
			nErrorWarningCode := 0;
		            sMessage := 'Success: Mover added.';				
		ELSE
			nErrorWarningCode := +11;
		            sMessage := 'Warning: Mover already exists.';				
		END_IF

	ELSE
		nErrorWarningCode := -11;
		        sMessage := 'Error: Mover invalid';	
	END_IF
	
	IF nErrorWarningCode < 0 THEN
		AddMover := FALSE;
	ELSE
		AddMover := TRUE;
	END_IF
END_METHOD

METHOD AddPosition : BOOL
VAR_INPUT
	x 	: LREAL;
	y	: LREAL;	
END_VAR



	nPositionCount := nPositionCount +1;
	
	IF nPositionCount <= gc_nMoverCountConfigured THEN
	
		positionList[nPositionCount].x     := x;
		positionList[nPositionCount].y     := y;
		positionList[nPositionCount].valid := TRUE;

		nErrorWarningCode := 0;
		        sMessage := 'Success: Position added.';				
	ELSE
		nPositionCount := gc_nMoverCountConfigured;	
	
		nErrorWarningCode := -21;
		        sMessage := 'Error: Position count higher than mover count!';				
	END_IF

	IF nErrorWarningCode < 0 THEN
		AddPosition := FALSE;
	ELSE
		AddPosition := TRUE;
	END_IF
END_METHOD

METHOD Clear : BOOL
VAR_INPUT
END_VAR




	FOR idx:=1 TO gc_nMoverCountConfigured DO
		MoverList[idx] := 0;
		
		positionList[idx].x     := 0;
		positionList[idx].y     := 0;
		positionList[idx].valid := FALSE;
		
	END_FOR	
	
	    nMoversInList := 0;
	   nPositionCount := 0;	
	       nStateMove := 0;
	nErrorWarningCode := 0;
			sMessage := 'Cleared';				

	Clear := TRUE;
END_METHOD

METHOD MoversToTarget : BOOL
VAR_INPUT
END_VAR



VAR_INST
	
	idx1, idx2						: UDINT;
	idxMover, idxPosition			: UDINT;
	fShortestDistance				: LREAL;
	targetPosition					: PositionXYC;
	currentPos						: PositionXYC;
	bDone							: BOOL;	
	
	fMoverDistanceToInitialPosition	: ARRAY [1..gc_nMoverCountConfigured, 1..gc_nMoverCountConfigured] OF ST_MoverDistance;   // Mover;Position
	nMoverToInitialPosition			: ARRAY [1..gc_nMoverCountConfigured] OF UDINT;
	nInitialPositionTakesMover		: ARRAY [1..gc_nMoverCountConfigured] OF UDINT;
	
	nInitialPositionTaken			: ARRAY [1..gc_nMoverCountConfigured] OF BOOL;	
	nInitialMoverTaken				: ARRAY [1..gc_nMoverCountConfigured] OF BOOL;	
	nMoverTaken						: UDINT;
	
	fShiftDistanceY			: LREAL := 240.0;
	fShiftDistanceX			: LREAL := 240.0;
	
	
	nTestCounter03	: UINT;
	nTestCounter01	: UINT;
	
	nMoveStatus						: ARRAY [1..gc_nMoverCountConfigured] OF DINT;	
	
	bMoverDone_01  					: BOOL;
	bMoverError_01 					: BOOL;
	bMoverDoneXYC_01  					: BOOL;
	bMoverErrorxyc_01 					: BOOL;

	
	bMoverDone_02  					: BOOL;
	bMoverError_02 					: BOOL;	
	bMoverDoneXYC_02  					: BOOL;
	bMoverErrorxyc_02 					: BOOL;
	
	stMoveToPositionOptions				: ST_MoveToPositionOptions;
	
	bStepByStep						: BOOL;
	bNextStep						: BOOL;
	
END_VAR
	
	CASE nStateMove OF 
		
	0:	// Check mover and position count
		IF nMoversInList <= nPositionCount THEN
			nErrorWarningCode := 0;
			        sMessage := 'Mover and position count OK.';	
			      nStateMove := nStateMove + 10;
		ELSE
			nErrorWarningCode := -31;
					sMessage := 'Error: Mover count higher than position count!';				
		END_IF
	
		
	10:	// Clear 
		FOR idx:=1 TO gc_nMoverCountConfigured DO
			        nMoveStatus[idx] := 0;
			 nInitialMoverTaken[idx] := 0;
		END_FOR	
		nStateMove := nStateMove + 10;
		
	
	20: // Calculate all distances
		FOR idx1:=1 TO gc_nMoverCountConfigured DO
			FOR idx2:=1 TO gc_nMoverCountConfigured DO
				fMoverDistanceToInitialPosition[idx1, idx2].fDistance      := 0.0;
				fMoverDistanceToInitialPosition[idx1, idx2].nPositionIndex := 0;
			END_FOR
		END_FOR
	
	
		FOR idx1:=1 TO nMoversInList DO
			currentPos.SetValuesXYC(moverList[idx1].std.P_SetPosition.x, moverList[idx1].std.P_SetPosition.y, moverList[idx1].std.P_SetPosition.c);
			FOR idx2:=1 TO nPositionCount DO
				fMoverDistanceToInitialPosition[idx1, idx2].nPositionIndex := idx2;		
				fMoverDistanceToInitialPosition[idx1, idx2].fDistance := SQRT((currentPos.x - positionList[idx2].x) * (currentPos.x - positionList[idx2].x) + (currentPos.y - positionList[idx2].y) * (currentPos.y - positionList[idx2].y)); 
			END_FOR	
			
			nInitialPositionTaken[idx1] := FALSE;
		END_FOR			

		nErrorWarningCode := 0;
				sMessage := 'Calculated all distances.';			
		      nStateMove := nStateMove + 10;
	
		
	30: // Find the closest initial position for each mover	
		FOR idxPosition:=1 TO nPositionCount DO
			fShortestDistance := 1.7976931348623158E+308;
			FOR idxMover:=1 TO nMoversInList DO			
				IF NOT nInitialMoverTaken[idxMover] THEN
					IF fMoverDistanceToInitialPosition[idxMover, idxPosition].fDistance < fShortestDistance THEN
						fShortestDistance := fMoverDistanceToInitialPosition[idxMover, idxPosition].fDistance;
						nInitialPositionTakesMover[idxPosition] := idxMover;
						nMoverTaken := idxMover;
					END_IF
				END_IF
			END_FOR
			IF nMoverTaken > 0 THEN
				nInitialMoverTaken[nMoverTaken] := TRUE;
			END_IF
		END_FOR
		
		
		FOR idx:=1 TO gc_nMoverCountConfigured DO
			nMoverToInitialPosition[nInitialPositionTakesMover[idx]] := idx;	
		END_FOR

		nErrorWarningCode := 0;
				sMessage := 'Calculated closest initial position for each mover.';			
		nStateMove := nStateMove + 10;
		
		
		
	40: // Turn all movers back to 0° 
		
		// -> warten auf Set-C rotation Feature aus der NC
			
		nStateMove := nStateMove + 10;
		
		
		
	50: // Moving all movers to their initial position

		nErrorWarningCode := 0;
				sMessage := 'Moving.';


		FOR idx1:=1 TO nMoversInList DO
			
			// 1st: try direct move
			IF  nMoveStatus[idx1] = 0 THEN
				currentPos.SetValuesXYC(moverList[idx1].std.P_SetPosition.x, moverList[idx1].std.P_SetPosition.y, moverList[idx1].std.P_SetPosition.c);
				targetPosition.SetValuesXYC(positionList[nMoverToInitialPosition[idx1]].x, positionList[nMoverToInitialPosition[idx1]].y, currentPos.c);
				stMoveToPositionOptions.useOrientation := FALSE;	
				IF moverList[idx1].std.MoveToPositionExt('ToTarget move direct', targetPosition, recoverVelocity, recoveryAcceleration, recoveryAcceleration, recoveryJerk, stMoveToPositionOptions) THEN
					nMoveStatus[idx1] := 1;
					IF bStepByStep THEN nMoveStatus[idx1] := -nMoveStatus[idx1]; END_IF
				END_IF
			END_IF
			
			// 2nd: try direct move XYC
			IF  nMoveStatus[idx1] = 1 THEN
				IF moverList[idx1].std.P_MoveToPositionExt.Error THEN
					currentPos.SetValuesXYC(moverList[idx1].std.P_SetPosition.x, moverList[idx1].std.P_SetPosition.y, moverList[idx1].std.P_SetPosition.c);
					targetPosition.SetValuesXYC(positionList[nMoverToInitialPosition[idx1]].x, positionList[nMoverToInitialPosition[idx1]].y, currentPos.c);
					stMoveToPositionOptions.useOrientation := TRUE;
					moverList[idx1].std.MoveToPositionExt('ToTarget move direct', targetPosition, recoverVelocity, recoveryAcceleration, recoveryAcceleration, recoveryJerk, stMoveToPositionOptions);
					nMoveStatus[idx1] := 2;
					IF bStepByStep THEN nMoveStatus[idx1] := -nMoveStatus[idx1]; END_IF
				END_IF
			END_IF			
			
			// 3rd: try move in x-direction
			IF  nMoveStatus[idx1] = 2 THEN
				IF moverList[idx1].std.P_MoveToPositionExt.Error THEN
					IF moverList[idx1].std.P_SetPosition.x <> positionList[nMoverToInitialPosition[idx1]].x THEN
						currentPos.SetValuesXYC(moverList[idx1].std.P_SetPosition.x, moverList[idx1].std.P_SetPosition.y, moverList[idx1].std.P_SetPosition.c);
						targetPosition.SetValuesXYC(positionList[nMoverToInitialPosition[idx1]].x, currentPos.y, currentPos.c);
						stMoveToPositionOptions.useOrientation := FALSE;
						moverList[idx1].std.MoveToPositionExt('ToTarget move in x', targetPosition, recoverVelocity, recoveryAcceleration, recoveryAcceleration, recoveryJerk, stMoveToPositionOptions);
					END_IF
					nMoveStatus[idx1] := 3;
					IF bStepByStep THEN nMoveStatus[idx1] := -nMoveStatus[idx1]; END_IF
				END_IF
			END_IF
						
			// 4th: try move XYC in x-direction
			IF  nMoveStatus[idx1] = 3 THEN
				IF moverList[idx1].std.P_MoveToPositionExt.Error THEN
					IF moverList[idx1].std.P_SetPosition.x <> positionList[nMoverToInitialPosition[idx1]].x THEN
						currentPos.SetValuesXYC(moverList[idx1].std.P_SetPosition.x, moverList[idx1].std.P_SetPosition.y, moverList[idx1].std.P_SetPosition.c);
						targetPosition.SetValuesXYC(positionList[nMoverToInitialPosition[idx1]].x, currentPos.y, currentPos.c);
						stMoveToPositionOptions.useOrientation := TRUE;
						moverList[idx1].std.MoveToPositionExt('ToTarget move in x', targetPosition, recoverVelocity, recoveryAcceleration, recoveryAcceleration, recoveryJerk, stMoveToPositionOptions);
					END_IF					
					nMoveStatus[idx1] := 4;
					IF bStepByStep THEN nMoveStatus[idx1] := -nMoveStatus[idx1]; END_IF
				END_IF
			END_IF			
			
			// 5th: try move in y-direction
			IF  nMoveStatus[idx1] = 4 THEN
				IF moverList[idx1].std.P_MoveToPositionExt.Error THEN
					IF moverList[idx1].std.P_SetPosition.y <> positionList[nMoverToInitialPosition[idx1]].y THEN
						currentPos.SetValuesXYC(moverList[idx1].std.P_SetPosition.x, moverList[idx1].std.P_SetPosition.y, moverList[idx1].std.P_SetPosition.c);
						targetPosition.SetValuesXYC(currentPos.x, positionList[nMoverToInitialPosition[idx1]].y, currentPos.c);
						stMoveToPositionOptions.useOrientation := FALSE;
						moverList[idx1].std.MoveToPositionExt('ToTarget move in y', targetPosition, recoverVelocity, recoveryAcceleration, recoveryAcceleration, recoveryJerk, stMoveToPositionOptions);
					END_IF
					nMoveStatus[idx1] := 5; 
					IF bStepByStep THEN nMoveStatus[idx1] := -nMoveStatus[idx1]; END_IF
				END_IF		
			END_IF			
			
			// 6th: try move XYC in y-direction
			IF  nMoveStatus[idx1] = 5 THEN
				IF moverList[idx1].std.P_MoveToPositionExt.Error THEN
					IF moverList[idx1].std.P_SetPosition.y <> positionList[nMoverToInitialPosition[idx1]].y THEN
						currentPos.SetValuesXYC(moverList[idx1].std.P_SetPosition.x, moverList[idx1].std.P_SetPosition.y, moverList[idx1].std.P_SetPosition.c);
						targetPosition.SetValuesXYC(currentPos.x, positionList[nMoverToInitialPosition[idx1]].y, currentPos.c);
						stMoveToPositionOptions.useOrientation := TRUE;
						moverList[idx1].std.MoveToPositionExt('ToTarget move in y', targetPosition, recoverVelocity, recoveryAcceleration, recoveryAcceleration, recoveryJerk, stMoveToPositionOptions);
					END_IF
					nMoveStatus[idx1] := 6; 
					IF bStepByStep THEN nMoveStatus[idx1] := -nMoveStatus[idx1]; END_IF
				END_IF		
			END_IF				
			
			// 7th: try positive step-move in y-direction
			IF  nMoveStatus[idx1] = 6 THEN
				IF moverList[idx1].std.P_MoveToPositionExt.Error THEN
					currentPos.SetValuesXYC(moverList[idx1].std.P_SetPosition.x, moverList[idx1].std.P_SetPosition.y, moverList[idx1].std.P_SetPosition.c);
					targetPosition.SetValuesXYC(currentPos.x, currentPos.y + fShiftDistanceY, currentPos.c);
					stMoveToPositionOptions.useOrientation := FALSE;
					moverList[idx1].std.MoveToPositionExt('ToTarget step-move in +y', targetPosition, recoverVelocity, recoveryAcceleration, recoveryAcceleration, recoveryJerk, stMoveToPositionOptions);
					nMoveStatus[idx1] := 7;
					IF bStepByStep THEN nMoveStatus[idx1] := -nMoveStatus[idx1]; END_IF
				END_IF		
			END_IF					
			
			// 8th: try positive step-move XYC in y-direction
			IF  nMoveStatus[idx1] = 7 THEN
				IF moverList[idx1].std.P_MoveToPositionExt.Error THEN
					currentPos.SetValuesXYC(moverList[idx1].std.P_SetPosition.x, moverList[idx1].std.P_SetPosition.y, moverList[idx1].std.P_SetPosition.c);
					targetPosition.SetValuesXYC(currentPos.x, currentPos.y + fShiftDistanceY, currentPos.c);
					stMoveToPositionOptions.useOrientation := TRUE;
					moverList[idx1].std.MoveToPositionExt('ToTarget step-move in +y', targetPosition, recoverVelocity, recoveryAcceleration, recoveryAcceleration, recoveryJerk, stMoveToPositionOptions);
					nMoveStatus[idx1] := 8; 
					IF bStepByStep THEN nMoveStatus[idx1] := -nMoveStatus[idx1]; END_IF
				END_IF		
			END_IF			
			
			// 9th: try negative step-move in y-direction
			IF  nMoveStatus[idx1] = 8 THEN
				IF moverList[idx1].std.P_MoveToPositionExt.Error THEN
					currentPos.SetValuesXYC(moverList[idx1].std.P_SetPosition.x, moverList[idx1].std.P_SetPosition.y, moverList[idx1].std.P_SetPosition.c);
					targetPosition.SetValuesXYC(currentPos.x, currentPos.y - fShiftDistanceX, currentPos.c);
					stMoveToPositionOptions.useOrientation := FALSE;
					moverList[idx1].std.MoveToPositionExt('ToTarget step-move in -y', targetPosition, recoverVelocity, recoveryAcceleration, recoveryAcceleration, recoveryJerk, stMoveToPositionOptions);
					nMoveStatus[idx1] := 9; 
					IF bStepByStep THEN nMoveStatus[idx1] := -nMoveStatus[idx1]; END_IF
				END_IF		
			END_IF	

			// 10th: try negative step-move XYC in y-direction
			IF  nMoveStatus[idx1] = 9 THEN 
				IF moverList[idx1].std.P_MoveToPositionExt.Error THEN
					currentPos.SetValuesXYC(moverList[idx1].std.P_SetPosition.x, moverList[idx1].std.P_SetPosition.y, moverList[idx1].std.P_SetPosition.c);
					targetPosition.SetValuesXYC(currentPos.x, currentPos.y - fShiftDistanceX, currentPos.c);
					stMoveToPositionOptions.useOrientation := TRUE;
					moverList[idx1].std.MoveToPositionExt('ToTarget step-move in -y', targetPosition, recoverVelocity, recoveryAcceleration, recoveryAcceleration, recoveryJerk, stMoveToPositionOptions);
					nMoveStatus[idx1] := 10; 
					IF bStepByStep THEN nMoveStatus[idx1] := -nMoveStatus[idx1]; END_IF
				END_IF		
			END_IF		

			// 11th: try positive step-move in x-direction
			IF  nMoveStatus[idx1] = 10 THEN
				IF moverList[idx1].std.P_MoveToPositionExt.Error THEN
					currentPos.SetValuesXYC(moverList[idx1].std.P_SetPosition.x, moverList[idx1].std.P_SetPosition.y, moverList[idx1].std.P_SetPosition.c);
					targetPosition.SetValuesXYC(currentPos.x  + fShiftDistanceY, currentPos.y, currentPos.c);
					stMoveToPositionOptions.useOrientation := FALSE;
					moverList[idx1].std.MoveToPositionExt('ToTarget step-move in +x', targetPosition, recoverVelocity, recoveryAcceleration, recoveryAcceleration, recoveryJerk, stMoveToPositionOptions);
					nMoveStatus[idx1] := 11; 
					IF bStepByStep THEN nMoveStatus[idx1] := -nMoveStatus[idx1]; END_IF
				END_IF		
			END_IF	
			
			// 12th: try positive step-move XYC in x-direction
			IF  nMoveStatus[idx1] = 11 THEN
				IF moverList[idx1].std.P_MoveToPositionExt.Error THEN
					currentPos.SetValuesXYC(moverList[idx1].std.P_SetPosition.x, moverList[idx1].std.P_SetPosition.y, moverList[idx1].std.P_SetPosition.c);
					targetPosition.SetValuesXYC(currentPos.x  + fShiftDistanceY, currentPos.y, currentPos.c);
					stMoveToPositionOptions.useOrientation := TRUE;
					moverList[idx1].std.MoveToPositionExt('ToTarget step-move in +x', targetPosition, recoverVelocity, recoveryAcceleration, recoveryAcceleration, recoveryJerk, stMoveToPositionOptions);
					nMoveStatus[idx1] := 12; 
					IF bStepByStep THEN nMoveStatus[idx1] := -nMoveStatus[idx1]; END_IF
				END_IF		
			END_IF					
			
			// 13th: try negative step-move in x-direction
			IF  nMoveStatus[idx1] = 12 THEN
				IF moverList[idx1].std.P_MoveToPositionExt.Error THEN
					currentPos.SetValuesXYC(moverList[idx1].std.P_SetPosition.x, moverList[idx1].std.P_SetPosition.y, moverList[idx1].std.P_SetPosition.c);
					targetPosition.SetValuesXYC(currentPos.x - fShiftDistanceY, currentPos.y, currentPos.c);
					stMoveToPositionOptions.useOrientation := FALSE;
					moverList[idx1].std.MoveToPositionExt('ToTarget step-move in -x', targetPosition, recoverVelocity, recoveryAcceleration, recoveryAcceleration, recoveryJerk, stMoveToPositionOptions);
					nMoveStatus[idx1] := 13; 
					IF bStepByStep THEN nMoveStatus[idx1] := -nMoveStatus[idx1]; END_IF
				END_IF		
			END_IF				
			
			// 14th: try negative step-move XYC in x-direction
			IF  nMoveStatus[idx1] = 13 THEN 
				IF moverList[idx1].std.P_MoveToPositionExt.Error THEN
					currentPos.SetValuesXYC(moverList[idx1].std.P_SetPosition.x, moverList[idx1].std.P_SetPosition.y, moverList[idx1].std.P_SetPosition.c);
					targetPosition.SetValuesXYC(currentPos.x - fShiftDistanceY, currentPos.y, currentPos.c);
					stMoveToPositionOptions.useOrientation := TRUE;
					moverList[idx1].std.MoveToPositionExt('ToTarget step-move in -x', targetPosition, recoverVelocity, recoveryAcceleration, recoveryAcceleration, recoveryJerk, stMoveToPositionOptions);
					nMoveStatus[idx1] := 0; 
					IF bStepByStep THEN nMoveStatus[idx1] := -nMoveStatus[idx1]; END_IF
				END_IF		
			END_IF				
			
			
			// Check feedback
			IF nMoveStatus[idx1] = 1
			OR nMoveStatus[idx1] = 2
			THEN
				IF moverList[idx1].std.P_MoveToPositionExt.Done THEN
					nMoveStatus[idx1] := 100;
				END_IF
			ELSE
				IF nMoveStatus[idx1] <> 100 THEN						
					// If y-move is finished or no move was possible
					IF moverList[idx1].std.P_MoveToPositionExt.Done THEN
						nMoveStatus[idx1] := 0;
					END_IF						
				END_IF
			END_IF
			
		END_FOR
		
	
		// Check if all movers have reached their position
		bDone := TRUE;
		FOR idx1:=1 TO nMoversInList DO
			IF nMoveStatus[idx1] <> 100 THEN
				bDone := FALSE;
			END_IF
		END_FOR
			
		IF bDone THEN
			nStateMove := nStateMove + 10;
		END_IF
		

	60: // Done
		nErrorWarningCode := 0;
				sMessage := 'Done';			
	
		   nStateMove := 0;
		MoversToTarget := TRUE;
			
	END_CASE
	
	
	
	IF bNextStep THEN
		bNextStep := FALSE;
		FOR idx1:=1 TO g_nMoverCountPresent DO
			nMoveStatus[idx1] := ABS(nMoveStatus[idx1]);
		END_FOR
	END_IF
END_METHOD

PROPERTY P_ErrorWarningCode : DINT
GET
P_ErrorWarningCode := nErrorWarningCode;
END_GET
END_PROPERTY

PROPERTY P_Info : STRING
GET
P_Info := sMessage;
END_GET
END_PROPERTY

PROPERTY P_ShiftDistanceX : LREAL
GET
P_ShiftDistanceX := fShiftDistanceX;
END_GET
SET
fShiftDistanceX := P_ShiftDistanceX;
END_SET
END_PROPERTY

PROPERTY P_ShiftDistanceY : LREAL
GET
P_ShiftDistanceY := fShiftDistanceY;
END_GET
SET
fShiftDistanceY := P_ShiftDistanceY;
END_SET
END_PROPERTY

METHOD SetDynamics : BOOL
VAR_INPUT
	vel	: LREAL;
	acc : LREAL;
	jerk :LREAL;
END_VAR

	recoverVelocity := vel;
	recoveryAcceleration := acc;
	recoveryJerk := jerk;
	
	SetDynamics := TRUE;
END_METHOD

END_FUNCTION_BLOCK

// ---- 2_Application/Mover/FB_ApplicationMover.TcPOU
FUNCTION_BLOCK FB_ApplicationMover IMPLEMENTS I_MoverApplication
VAR
	ipMoverStandard	: I_XPlanarMoverStandard;
	
	stProductData	: ST_ProductData;
	
	nMoverIndex		: INT;
	
	nTrackId		: UDINT;
	
	// customer Data
	bIsLoaded		: BOOL;	
		
				
END_VAR

VAR_OUTPUT
	VisuPos	: MoverVector;
END_VAR

METHOD Cycle


VAR_INST
	nTestCounter	: UINT;
END_VAR
IF std <> 0 THEN
	
	nTestCounter := nTestCounter +1;
	
	std.cycle();
	
	VisuPos   := std.P_ActPosition;
	VisuPos.c := std.P_RotationAngleModulo;
			
END_IF
END_METHOD

PROPERTY P_MoverIndex : INT
GET
P_MoverIndex := nMoverIndex;
END_GET
SET
nMoverIndex := P_MoverIndex;
END_SET
END_PROPERTY

PROPERTY P_ProductData : Reference to ST_ProductData
GET
P_ProductData REF= stProductData;
END_GET
SET
stProductData := P_ProductData;
END_SET
END_PROPERTY

PROPERTY P_TrackId : UDINT
GET
P_TrackId := nTrackId;
END_GET
SET
nTrackId := P_TrackId;
END_SET
END_PROPERTY

PROPERTY std : I_XPlanarMoverStandard
GET
IF ipMoverStandard <> 0 THEN
	std := ipMoverStandard;	
END_IF
END_GET
SET
ipMoverStandard := std;
END_SET
END_PROPERTY

END_FUNCTION_BLOCK

// ---- VISU/Logic/FB_VisuMessage.TcPOU
FUNCTION_BLOCK FB_VisuMessage IMPLEMENTS I_VisuMessage;


VAR	
	bInfo				: BOOL;
	bAlarm				: BOOL;
	bError				: BOOL;

	nMessageColor		: DWORD;
	_sMessageText_L1	: STRING;
	_sMessageText_L2	: STRING;

	stVisuOut			: ST_VisuMessage;


	sInfoMessage		: STRING;
	sInfoSequence		: STRING;
	nInfoState			: DINT;
	
	sCurrentSequence	: STRING;
	
	_sErrorMessage	: STRING;
	_sErrorSequence	: STRING;
	_nErrorState	: DINT;
	_nErrorCode		: DWORD;

	nColor_Green	: DWORD := 16#FF189E00;
	nColor_Yellow	: DWORD := 16#FFE6A000;
	nColor_Red		: DWORD := 16#FFFF0000;
	nColor_Black	: DWORD := 16#FF000000;


	_bAcknowledge	: BOOL;
	
	
	
END_VAR

METHOD CheckAknowledge : BOOL
VAR_INPUT
END_VAR



	CheckAknowledge := _bAcknowledge;
	  _bAcknowledge := FALSE;
END_METHOD

METHOD ClearAlarmMessage : BOOL
VAR_INPUT
END_VAR
END_METHOD

METHOD ClearAllMessages : BOOL
VAR_INPUT
END_VAR

	bError := FALSE;
	bInfo  := FALSE;
	
	ClearAllMessages := TRUE;
END_METHOD

METHOD ClearInfoMessage : BOOL
VAR_INPUT
END_VAR



	bInfo  := FALSE;
	
	ClearInfoMessage := TRUE;
END_METHOD

METHOD Cycle : BOOL
VAR_INPUT
	bAcknowledge	: BOOL;
END_VAR


	IF bAcknowledge THEN
		_bAcknowledge := TRUE;
	END_IF


	stVisuOut.bVisible_Box1_A := FALSE;
	stVisuOut.bVisible_Box1_B := FALSE;		


	IF bInfo THEN
		_sMessageText_L1 := CONCAT(sInfoMessage, ' - ');
		_sMessageText_L1 := CONCAT(_sMessageText_L1, sInfoSequence);
		
		IF nInfoState <> 0 THEN	
			_sMessageText_L1 := CONCAT(_sMessageText_L1, ' - State:');
			_sMessageText_L1 := CONCAT(_sMessageText_L1, DINT_TO_STRING(nInfoState));
		END_IF
		
		stVisuOut.bVisible_Box1_A := TRUE;
		stVisuOut.bVisible_Box1_B := FALSE;		
		
		stVisuOut.sMessage_L1_Box1.sText  := _sMessageText_L1;
		stVisuOut.sMessage_L1_Box1.nColor := nColor_Green;
	END_IF
	
	
	
//	IF bAlarm THEN
//		stVisuOut.sMessage_L1_Box1 := _sMessageText_L1;
//		stVisuOut.nColor_Box1   := nColor_Yellow;
//	END_IF

	
	
	
	IF bError THEN
		
		_sMessageText_L1 := CONCAT('Sequence: ' , _sErrorSequence);
		_sMessageText_L1 := CONCAT(_sMessageText_L1, ' - State:');
		_sMessageText_L1 := CONCAT(_sMessageText_L1, DINT_TO_STRING(_nErrorState));	
		

		_sMessageText_L2 := CONCAT('Error Message: ', _sErrorMessage);
		
		IF _nErrorCode > 0 THEN 
			_sMessageText_L2 := CONCAT(_sMessageText_L2,  ' - Error Code: ');
			_sMessageText_L2 := CONCAT(_sMessageText_L2, DWORD_TO_STRING(_nErrorCode));
		END_IF
	
	
		stVisuOut.bVisible_Box1_A := FALSE;
		stVisuOut.bVisible_Box1_B := TRUE;

		
		stVisuOut.sMessage_L1_Box1.sText  := _sMessageText_L1;
		stVisuOut.sMessage_L1_Box1.nColor := nColor_Red;
		
		stVisuOut.sMessage_L2_Box1.sText  := _sMessageText_L2;
		stVisuOut.sMessage_L2_Box1.nColor := nColor_Red;
		
	END_IF
END_METHOD

PROPERTY P_VisuOut : ST_VisuMessage
GET
P_VisuOut := stVisuOut;
END_GET
END_PROPERTY

METHOD SetAlarmMessage : BOOL
VAR_INPUT
	sMessage	: STRING;
END_VAR



	bError := FALSE;

	SetAlarmMessage := TRUE;
END_METHOD

METHOD SetErrorMessage : BOOL
VAR_INPUT
	sMessage	: STRING;
	sSequence	: STRING;
	nState		: DINT;
	nErrorCode	: DWORD;
END_VAR

	bError := TRUE;
	bInfo  := FALSE;

	_sErrorMessage	:= sMessage;
	_sErrorSequence	:= sSequence;
	
	sCurrentSequence := sSequence;
	
	_nErrorState	:= nState;
	_nErrorCode		:= nErrorCode;
	
	
	SetErrorMessage := TRUE;
END_METHOD

METHOD SetInfoMessage : BOOL
VAR_INPUT
	sMessage	: STRING;
	sSequence	: STRING;
	nState		: DINT;
END_VAR

	bInfo  := TRUE;
	bError := FALSE;

	
	sInfoMessage	 := sMessage;
	sInfoSequence	 := sSequence;
	sCurrentSequence := sSequence;
	nInfoState		 := nState;
	
	
	SetInfoMessage  := TRUE;
END_METHOD

METHOD StateUpdate : BOOL
VAR_INPUT
	nState		: DINT;
	sSequence	: STRING;
END_VAR



	IF sSequence = sCurrentSequence THEN

		nInfoState := nState;
		
	END_IF



	
	StateUpdate := TRUE;
END_METHOD

END_FUNCTION_BLOCK

// ---- 2_Application/Tracks/FB_TrackSegment_1.TcPOU
FUNCTION_BLOCK FB_TrackSegment_1 EXTENDS FB_TrackBase IMPLEMENTS I_TRACK
VAR_INPUT
END_VAR
VAR_OUTPUT
END_VAR

METHOD Initialize : BOOL
VAR_INPUT
	nTrackIndex : UDINT;
END_VAR

VAR_INST
	TrackTable		: FB_TrackTable;
	
	nPointIndex		: INT;
	nPointIndexA	: INT;	
	nPointIndexB	: INT;	
	idx1, idx2		: INT;
	nStartFromTrack	: INT;
	nEndAtTrack		: INT;
	bCloseLoop		: BOOL;	
	
	bTrackBuild		: BOOL;
	StartFromTrack	: I_Track;
	EndAtTrack		: I_Track;
	
	sIndexWhereTheCheckFailed	: UINT;
	nErrorID					: UDINT;

END_VAR





VAR_INST
	
	TrackTableTemp		: ARRAY[1..gc_MaxNumberTrackPoints] OF ST_TrackTable;
	


END_VAR


VAR_INST
	
	pos01	:		PositionXYC;
	pos02	:		PositionXYC;


END_VAR

	  
CASE nState OF 

	10:	// Starting with an empty table. 
		IF TrackTable.ClearTrackTable() THEN
			nState := nState + 10;
		END_IF
		

	20:	// Init Track-Table
		
		// *************************************************************************************
		// *** Only the code in this state must be eddited according to machine/track layout ***
		// *************************************************************************************	
		
		nStartFromTrack	:= 0;		// 0 for the first track all others according to their predecessor!
	    	nEndAtTrack := 0;		// 0 for the first track all others according to their successor! 		
		     bCloseLoop := FALSE;	// TRUE for circular track	

			 			 			 
		// Building the track table:	
		TrackTable.AddPoint(E_PointType.Line_Start, E_PointOption.none, 480.0, 120.0, 0.0); 	 
		TrackTable.AddPoint(E_PointType.Line_End,   E_PointOption.none, 240.0, 120.0, 0.0);				
		
		TrackTable.AddPoint(E_PointType.Line_Start, E_PointOption.none, 120.0, 240.0, 0.0); 	 
		TrackTable.AddPoint(E_PointType.Line_End,   E_PointOption.none, 120.0, 480.0, 0.0);	
 
		TrackTable.AddPoint(E_PointType.Line_Start, E_PointOption.none, 240.0, 600.0, 0.0); 	 
		TrackTable.AddPoint(E_PointType.Line_End,   E_PointOption.none, 480.0, 600.0, 0.0);		
	 		
		nState := nState + 10;


	30:
		// *************************************************************
		// ***       NO Code Changes are needed from here on!        ***
		// *************************************************************		
			
		// The track table contains all additional information, too.
		IF nStartFromTrack > 0 THEN
			TrackTable.P_StartFromTrack := ipTrack[nStartFromTrack].std;	
		END_IF
		IF nEndAtTrack > 0 THEN
			TrackTable.P_EndAtTrack := ipTrack[nEndAtTrack].std;	
		END_IF	
		TrackTable.P_CloseTheLoop := bCloseLoop;	
		nState := nState + 10;

			
		
	40: // Checking the track table for plausibility
		IF TrackTable.CheckTrackTable() <> 0 THEN
			IF TrackTable.P_TrackTableCheckResult THEN
				nState := 50;	// Plausibility test succeeded.
			ELSE
				nState := 41;	// Plausibility test failed!
			END_IF
		END_IF

	
	41:	// In case of failed plausibility test check the creation of the above track table.
		// A Line must always begin with E_PointType.Line_Start and end with E_PointType.Line_End.
		// A Circle must always be added in the order E_PointType.Circle_Start, E_PointType.Circle_Center, E_PointType.Circle_End.
		// Check the info text for further information:
		sErrorInfoTextTemp := CONCAT('Track: ', UDINT_TO_STRING(nTrackIndex));
		sErrorInfoTextTemp := CONCAT(sErrorInfoTextTemp, ' - ');
		sErrorInfoTextTemp := CONCAT(sErrorInfoTextTemp, TrackTable.P_InfoText);
		
				     bTrackBuildError := TRUE;
					   sErrorInfoText := sErrorInfoTextTemp;
			sIndexWhereTheCheckFailed := TrackTable.P_TrackCheckImplausibleTableIndex;
					   TrackTableTemp := TrackTable.P_Table;	
							
 					   
	50:	// Building the track	
		IF fbTrackStandard.BuildTrackExt(TrackTable) THEN
			nState := nState +1;
		END_IF
		
	51:	IF fbTrackStandard.P_BuildTrackExt.Done THEN
			nState := 100;	
		ELSIF fbTrackStandard.P_BuildTrackExt.Error THEN
	  		nState := nState +1;
		END_IF		
		
	52: // In case an error occured, check the error ID and InfoText and react accordingly:
		sErrorInfoTextTemp := CONCAT('Track: ', UDINT_TO_STRING(nTrackIndex));
		sErrorInfoTextTemp := CONCAT(sErrorInfoTextTemp, ' - ');
		sErrorInfoTextTemp := CONCAT(sErrorInfoTextTemp, fbTrackStandard.P_BuildTrackExtInfoText);	
	
			      nErrorID := fbTrackStandard.P_BuildTrackExt.ErrorID;
		    sErrorInfoText := sErrorInfoTextTemp;		
			
		  bTrackBuildError := TRUE;		   
					   
		 
	100: 	// Track build done
			fTrackLength := fbTrackStandard.GetLength();
			  Initialize := TRUE;
	

END_CASE
END_METHOD

PROPERTY P_Error : BOOL
GET
P_Error := bTrackBuildError;
END_GET
END_PROPERTY

PROPERTY P_ErrorInfo : STRING
GET
P_ErrorInfo := sErrorInfoText;
END_GET
END_PROPERTY

END_FUNCTION_BLOCK

// ---- 2_Application/Tracks/Base/FB_TrackBase.TcPOU
FUNCTION_BLOCK FB_TrackBase


VAR
	trackLinePosStart 	: PositionXYC;
	trackLinePosEnd 	: PositionXYC;
	fbTrackStandard		: FB_TrackStandard;
	fTrackLength		: LREAL;

	nState				: INT;
	sErrorInfoText		: STRING;
	sErrorInfoTextTemp	: STRING;
	bTrackBuildError	: BOOL;

END_VAR

METHOD Clear : BOOL


VAR_INST
	
	nStateReset		: UINT;

END_VAR


	CASE nStateReset OF
		
	0:	nStateReset := 10;
	
	10: IF fbTrackStandard.P_State = MC_PLANAR_STATE.Error
		OR fbTrackStandard.P_State = MC_PLANAR_STATE.ErrorPending
		THEN
			nStateReset := nStateReset +1;
		ELSE
			nStateReset := nStateReset +10;
		END_IF
		
	11: IF fbTrackStandard.Reset() THEN
			nStateReset := nStateReset +1;
		END_IF
	
	12:	IF fbTrackStandard.P_Reset.Done THEN
			nStateReset := nStateReset +8;
		END_IF
	
	20:
		  sErrorInfoText := '';
		bTrackBuildError := FALSE;
				  nState := 10;
				   Clear := TRUE;	
	
		nStateReset := 0;
	
	END_CASE
END_METHOD

METHOD Cycle : BOOL
VAR_INPUT
END_VAR
fbTrackStandard.Cycle();
END_METHOD

PROPERTY P_TrackLength : LREAL
GET
P_TrackLength := fTrackLength;
END_GET
END_PROPERTY

PROPERTY std : I_TrackStandard
GET
std := fbTrackStandard;
END_GET
END_PROPERTY

END_FUNCTION_BLOCK

// ---- 2_Application/Tracks/FB_TrackSegment_2.TcPOU
FUNCTION_BLOCK FB_TrackSegment_2 EXTENDS FB_TrackBase IMPLEMENTS I_TRACK
VAR_INPUT
END_VAR
VAR_OUTPUT
END_VAR

METHOD Initialize : BOOL

VAR_INPUT
	nTrackIndex : UDINT;
END_VAR


VAR_INST
	TrackTable		: FB_TrackTable;
	
	nPointIndex		: INT;
	nPointIndexA	: INT;	
	nPointIndexB	: INT;	
	idx1, idx2		: INT;
	nStartFromTrack	: INT;
	nEndAtTrack		: INT;
	bCloseLoop		: BOOL;	
	
	bTrackBuild		: BOOL;
	StartFromTrack	: I_Track;
	EndAtTrack		: I_Track;
	
	sIndexWhereTheCheckFailed	: UINT;
	nErrorID					: UDINT;

END_VAR





VAR_INST
	
	TrackTableTemp		: ARRAY[1..gc_MaxNumberTrackPoints] OF ST_TrackTable;
	


END_VAR


VAR_INST
	
	pos01	:		PositionXYC;
	pos02	:		PositionXYC;


END_VAR

	  
CASE nState OF 

	10:	// Starting with an empty table. 
		IF TrackTable.ClearTrackTable() THEN
			nState := nState + 10;
		END_IF
		

	20:	// Init Track-Table
		
		// *************************************************************************************
		// *** Only the code in this state must be eddited according to machine/track layout ***
		// *************************************************************************************	
		
		nStartFromTrack	:= 1;		// 0 for the first track all others according to their predecessor!
	    	nEndAtTrack := 1;		// 0 for the first track all others according to their successor! 		
		     bCloseLoop := FALSE;	// TRUE for circular track	

			 			 			 
		// Building the track table:
		TrackTable.AddPoint(E_PointType.Line_Start, E_PointOption.none, 600.0, 480.0, 0.0); 	 
		TrackTable.AddPoint(E_PointType.Line_End,   E_PointOption.none, 600.0, 240.0, 0.0);				
						
		nState := nState + 10;


	30:
		// *************************************************************
		// ***       NO Code Changes are needed from here on!        ***
		// *************************************************************		
			
		// The track table contains all additional information, too.
		IF nStartFromTrack > 0 THEN
			TrackTable.P_StartFromTrack := ipTrack[nStartFromTrack].std;	
		END_IF
		IF nEndAtTrack > 0 THEN
			TrackTable.P_EndAtTrack := ipTrack[nEndAtTrack].std;	
		END_IF	
		TrackTable.P_CloseTheLoop := bCloseLoop;	
		nState := nState + 10;

			
		
	40: // Checking the track table for plausibility
		IF TrackTable.CheckTrackTable() <> 0 THEN
			IF TrackTable.P_TrackTableCheckResult THEN
				nState := 50;	// Plausibility test succeeded.
			ELSE
				nState := 41;	// Plausibility test failed!
			END_IF
		END_IF

	
	41:	// In case of failed plausibility test check the creation of the above track table.
		// A Line must always begin with E_PointType.Line_Start and end with E_PointType.Line_End.
		// A Circle must always be added in the order E_PointType.Circle_Start, E_PointType.Circle_Center, E_PointType.Circle_End.
		// Check the info text for further information:
		sErrorInfoTextTemp := CONCAT('Track: ', UDINT_TO_STRING(nTrackIndex));
		sErrorInfoTextTemp := CONCAT(sErrorInfoTextTemp, ' - ');
		sErrorInfoTextTemp := CONCAT(sErrorInfoTextTemp, TrackTable.P_InfoText);
		
				     bTrackBuildError := TRUE;
					   sErrorInfoText := sErrorInfoTextTemp;
			sIndexWhereTheCheckFailed := TrackTable.P_TrackCheckImplausibleTableIndex;
					   TrackTableTemp := TrackTable.P_Table;	
							
 					   
	50:	// Building the track	
		IF fbTrackStandard.BuildTrackExt(TrackTable) THEN
			nState := nState +1;
		END_IF
		
	51:	IF fbTrackStandard.P_BuildTrackExt.Done THEN
			nState := 100;	
		ELSIF fbTrackStandard.P_BuildTrackExt.Error THEN
	  		nState := nState +1;
		END_IF		
		
	52: // In case an error occured, check the error ID and InfoText and react accordingly:
		sErrorInfoTextTemp := CONCAT('Track: ', UDINT_TO_STRING(nTrackIndex));
		sErrorInfoTextTemp := CONCAT(sErrorInfoTextTemp, ' - ');
		sErrorInfoTextTemp := CONCAT(sErrorInfoTextTemp, fbTrackStandard.P_BuildTrackExtInfoText);	
	
			      nErrorID := fbTrackStandard.P_BuildTrackExt.ErrorID;
		    sErrorInfoText := sErrorInfoTextTemp;		
			
		  bTrackBuildError := TRUE;		   
					   
		 
	100: 	// Track build done
			fTrackLength := fbTrackStandard.GetLength();
			  Initialize := TRUE;
	
			
END_CASE
END_METHOD

PROPERTY P_Error : BOOL
GET
P_Error := bTrackBuildError;
END_GET
END_PROPERTY

PROPERTY P_ErrorInfo : STRING
GET
P_ErrorInfo := sErrorInfoText;
END_GET
END_PROPERTY

END_FUNCTION_BLOCK

// ---- 2_Application/Tracks/FB_TrackSegment_3.TcPOU
FUNCTION_BLOCK FB_TrackSegment_3 EXTENDS FB_TrackBase IMPLEMENTS I_TRACK
VAR_INPUT
END_VAR
VAR_OUTPUT
END_VAR

METHOD Initialize : BOOL

VAR_INPUT
	nTrackIndex : UDINT;
END_VAR


VAR_INST
	TrackTable		: FB_TrackTable;
	
	nPointIndex		: INT;
	nPointIndexA	: INT;	
	nPointIndexB	: INT;	
	idx1, idx2		: INT;
	nStartFromTrack	: INT;
	nEndAtTrack		: INT;
	bCloseLoop		: BOOL;	
	
	bTrackBuild		: BOOL;
	StartFromTrack	: I_Track;
	EndAtTrack		: I_Track;
	
	sIndexWhereTheCheckFailed	: UINT;
	nErrorID					: UDINT;

END_VAR





VAR_INST
	
	TrackTableTemp		: ARRAY[1..gc_MaxNumberTrackPoints] OF ST_TrackTable;
	


END_VAR


VAR_INST
	
	pos01	:		PositionXYC;
	pos02	:		PositionXYC;


END_VAR

	  
CASE nState OF 

	10:	// Starting with an empty table. 
		IF TrackTable.ClearTrackTable() THEN
			nState := nState + 10;
		END_IF
		

	20:	// Init Track-Table
		
		// *************************************************************************************
		// *** Only the code in this state must be eddited according to machine/track layout ***
		// *************************************************************************************	
		
		nStartFromTrack	:= 1;		// 0 for the first track all others according to their predecessor!
	    	nEndAtTrack := 1;		// 0 for the first track all others according to their successor! 		
		     bCloseLoop := FALSE;	// TRUE for circular track	

			 			 			 
		// Building the track table:
		TrackTable.AddPoint(E_PointType.Line_Start, E_PointOption.none, 480.0, 600.0, 0.0); 	 
		TrackTable.AddPoint(E_PointType.Line_End,   E_PointOption.none, 720.0, 600.0, 0.0);				
						
		TrackTable.AddPoint(E_PointType.Line_Start, E_PointOption.none, 840.0, 480.0, 0.0); 	 
		TrackTable.AddPoint(E_PointType.Line_End,   E_PointOption.none, 840.0, 240.0, 0.0);			
		
		TrackTable.AddPoint(E_PointType.Line_Start, E_PointOption.none, 720.0, 120.0, 0.0); 	 
		TrackTable.AddPoint(E_PointType.Line_End,   E_PointOption.none, 480.0, 120.0, 0.0);			
		
		nState := nState + 10;

		
	30:
		// *************************************************************
		// ***       NO Code Changes are needed from here on!        ***
		// *************************************************************		
			
		// The track table contains all additional information, too.
		IF nStartFromTrack > 0 THEN
			TrackTable.P_StartFromTrack := ipTrack[nStartFromTrack].std;	
		END_IF
		IF nEndAtTrack > 0 THEN
			TrackTable.P_EndAtTrack := ipTrack[nEndAtTrack].std;	
		END_IF	
		TrackTable.P_CloseTheLoop := bCloseLoop;	
		nState := nState + 10;

			
		
	40: // Checking the track table for plausibility
		IF TrackTable.CheckTrackTable() <> 0 THEN
			IF TrackTable.P_TrackTableCheckResult THEN
				nState := 50;	// Plausibility test succeeded.
			ELSE
				nState := 41;	// Plausibility test failed!
			END_IF
		END_IF

	
	41:	// In case of failed plausibility test check the creation of the above track table.
		// A Line must always begin with E_PointType.Line_Start and end with E_PointType.Line_End.
		// A Circle must always be added in the order E_PointType.Circle_Start, E_PointType.Circle_Center, E_PointType.Circle_End.
		// Check the info text for further information:
		sErrorInfoTextTemp := CONCAT('Track: ', UDINT_TO_STRING(nTrackIndex));
		sErrorInfoTextTemp := CONCAT(sErrorInfoTextTemp, ' - ');
		sErrorInfoTextTemp := CONCAT(sErrorInfoTextTemp, TrackTable.P_InfoText);
		
				     bTrackBuildError := TRUE;
					   sErrorInfoText := sErrorInfoTextTemp;
			sIndexWhereTheCheckFailed := TrackTable.P_TrackCheckImplausibleTableIndex;
					   TrackTableTemp := TrackTable.P_Table;	
							
 					   
	50:	// Building the track	
		IF fbTrackStandard.BuildTrackExt(TrackTable) THEN
			nState := nState +1;
		END_IF
		
	51:	IF fbTrackStandard.P_BuildTrackExt.Done THEN
			nState := 100;	
		ELSIF fbTrackStandard.P_BuildTrackExt.Error THEN
	  		nState := nState +1;
		END_IF		
		
	52: // In case an error occured, check the error ID and InfoText and react accordingly:
		sErrorInfoTextTemp := CONCAT('Track: ', UDINT_TO_STRING(nTrackIndex));
		sErrorInfoTextTemp := CONCAT(sErrorInfoTextTemp, ' - ');
		sErrorInfoTextTemp := CONCAT(sErrorInfoTextTemp, fbTrackStandard.P_BuildTrackExtInfoText);	
	
			      nErrorID := fbTrackStandard.P_BuildTrackExt.ErrorID;
		    sErrorInfoText := sErrorInfoTextTemp;		
			
		  bTrackBuildError := TRUE;		   
					   
		 
	100: 	// Track build done
			fTrackLength := fbTrackStandard.GetLength();
			  Initialize := TRUE;
	
			
END_CASE
END_METHOD

METHOD Initialize_Test : BOOL


VAR_INST
	TrackTable		: FB_TrackTable;
	
	nPointIndex		: INT;
	nPointIndexA	: INT;	
	nPointIndexB	: INT;	
	idx1, idx2		: INT;
	nStartFromTrack	: INT;
	nEndAtTrack		: INT;
	bCloseLoop		: BOOL;	
	
	bTrackBuild		: BOOL;
	StartFromTrack	: I_Track;
	EndAtTrack		: I_Track;
	
	sIndexWhereTheCheckFailed	: UINT;
	nErrorID					: UDINT;

END_VAR





VAR_INST
	
	TrackTableTemp		: ARRAY[1..maxNumTrackPoints] OF ST_TrackTable;
	


END_VAR


VAR_INST
	
	pos01	:		PositionXYC;
	pos02	:		PositionXYC;


END_VAR

	  
CASE nState OF 

	10:	// Starting with an empty table. 
		IF TrackTable.ClearTrackTable() THEN
			nState := nState + 10;
		END_IF
		

	20:	// Init Track-Table
		
		// *************************************************************************************
		// *** Only the code in this state must be eddited according to machine/track layout ***
		// *************************************************************************************	
		
		nStartFromTrack	:= 0;		// 0 for the first track all others according to their predecessor!
	    	nEndAtTrack := 0;		// 0 for the first track all others according to their successor! 		
		     bCloseLoop := TRUE;	// TRUE for circular track	

			 			 			 
		// Building the track table:
		TrackTable.AddPoint(E_PointType.Point, E_PointOption.none, 485.0, 605.0, 0.0); 	 
								
		TrackTable.AddPoint(E_PointType.Line_Start, E_PointOption.none, 490.0, 610.0, 0.0); 	 
		TrackTable.AddPoint(E_PointType.Line_End,   E_PointOption.none, 590.0, 690.0, 0.0);			
		 
		TrackTable.AddPoint(E_PointType.Circle_Start,  E_PointOption.none, 700.0, 700.0, 0.0);
		TrackTable.AddPoint(E_PointType.Circle_Center, E_PointOption.none, 700.0, 800.0, 0.0); 	 
		TrackTable.AddPoint(E_PointType.Circle_End,    E_PointOption.none, 700.0, 900.0, 0.0);			
		
		nState := nState + 10;

		
	30:
		// *************************************************************
		// ***       NO Code Changes are needed from here on!        ***
		// *************************************************************		
			
		// The track table contains all additional information, too.
		IF nStartFromTrack > 0 THEN
			TrackTable.P_StartFromTrack := ipTrack[nStartFromTrack].std;	
		END_IF
		IF nEndAtTrack > 0 THEN
			TrackTable.P_EndAtTrack := ipTrack[nEndAtTrack].std;	
		END_IF	
		TrackTable.P_CloseTheLoop := bCloseLoop;	
		nState := nState + 10;

			
		
	40: // Checking the track table for plausibility
		IF TrackTable.CheckTrackTable() <> 0 THEN
			IF TrackTable.P_TrackTableCheckResult THEN
				nState := 50;	// Plausibility test succeeded.
			ELSE
				nState := 41;	// Plausibility test failed!
			END_IF
		END_IF

	
	41:	// In case of failed plausibility test check the creation of the above track table.
		// A Line must always begin with E_PointType.Line_Start and end with E_PointType.Line_End.
		// A Circle must always be added in the order E_PointType.Circle_Start, E_PointType.Circle_Center, E_PointType.Circle_End.
		// Check the info text for further information:
				     bTrackBuildError := TRUE;
			           sErrorInfoText := TrackTable.P_InfoText;
			sIndexWhereTheCheckFailed := TrackTable.P_TrackCheckImplausibleTableIndex;
					   TrackTableTemp := TrackTable.P_Table;	
							
 			
	50:	// Building the track	
		IF fbTrackStandard.BuildTrackExt(TrackTable) THEN
			nState := nState +1;
		END_IF
		
	51:	IF fbTrackStandard.P_BuildTrackExt.Done THEN
			nState := 100;	
		ELSIF fbTrackStandard.P_BuildTrackExt.Error THEN
	  		nState := nState +1;
		END_IF		
		
	52: // In case an error occured, check the error ID and InfoText and react accordingly:
			      nErrorID := fbTrackStandard.P_BuildTrackExt.ErrorID;
		    sErrorInfoText := fbTrackStandard.P_BuildTrackExtInfoText;		
			
		  bTrackBuildError := TRUE;		   
					   
		 
	100: 	// Track build done
			fTrackLength := fbTrackStandard.GetLength();
			  Initialize := TRUE;
	
			
END_CASE
END_METHOD

PROPERTY P_Error : BOOL
GET
P_Error := bTrackBuildError;
END_GET
END_PROPERTY

PROPERTY P_ErrorInfo : STRING
GET
P_ErrorInfo := sErrorInfoText;
END_GET
END_PROPERTY

END_FUNCTION_BLOCK

// ---- 2_Application/Station/FB_Station_01_Process.TcPOU
FUNCTION_BLOCK FB_Station_01_Process EXTENDS FB_StationBase
VAR
	nStationIndex				: UINT;
	nNextStationIndex			: UINT;
	nStationTrackIndex			: UINT;
	
	fStationPosition_X 			: LREAL;
	fStationPosition_Y 			: LREAL;		  
    fSendAwayDistance			: LREAL;	
	fInRangeDistance			: LREAL;	
	fSendAwayPosition			: LREAL;
	
	position					: PositionXYC;

END_VAR

METHOD Clear : BOOL
VAR_INPUT
END_VAR



	CASE nStateClear OF
		
	0:	// Enter
		Clear := FALSE;
		nStateClear := nStateClear +10;
		
	10: // Clearing all Station-Lists 
		IF SUPER^.Clear() THEN
			nStateClear := nStateClear +10;
		END_IF	
	
	20:	// Add aditional Data to be cleared here...
		nStateClear := 100;
		
		
	100: // Done
		      Clear := TRUE;
		nStateClear := 0;

	END_CASE
END_METHOD

METHOD Init : BOOL



VAR_INST
	nTestCounter	: INT;	
END_VAR
nTestCounter := nTestCounter +1;

CASE nStateInit OF

	0:		// Enter 
			bStationInitDone := FALSE;
			   nStateProcess := 0;
			      nStateInit := 10;
				 
			
	10:		// Init Station-Parameters				
				  nStationIndex := 1;				// Each station needs an unique index	
			 nStationTrackIndex := 1;	 			// Track on which the station resides
			  nNextStationIndex := 4;				// Index of the following station 
							  
			 fStationPosition_X := 120.0;			// Position of the station in X/Y coordinates
			 fStationPosition_Y := 360.0;			// Position of the station in X/Y coordinates
			  
			  fSendAwayDistance := 300.0;			// Position on track a mover will be send to after processing 
			  fInRangeDistance  := 300.0;			// Position in front of a station from where a mover will be taken over
			  
			  nStateInit := 11;
				   
				  
	11: // Fail-safe check, just to make sure all variables have been assigned after doing copy&paste from the template
			IF        nStationIndex > 0
			AND  nStationTrackIndex > 0
			AND   nNextStationIndex > 0
			AND  fStationPosition_X > 0
			AND  fStationPosition_Y > 0
			AND   fSendAwayDistance > 0
			THEN   
				nStateInit := 20;
			END_IF
			
				   
	20:		// Calculating positions
	
			// 1. Calculating station position on track
			position.SetValuesXYC(fStationPosition_X, fStationPosition_Y, 0.0);
			fStationPositionOnTrack := ipTrack[nStationTrackIndex].std.GetTrackPositionAt(position);
							
			// 2. Calculating send-away position on track
			fSendAwayPosition := fStationPositionOnTrack + fSendAwayDistance; 
			
			// The send away position must not exceed the lenght of the track!
			IF fSendAwayPosition > ipTrack[nStationTrackIndex].P_TrackLength THEN
				fSendAwayPosition := ipTrack[nStationTrackIndex].P_TrackLength;
			END_IF
			
			// 3. Calculating the station position in X/Y coordinates determined by the track	
            //    This is to make sure the center of the station is always located directly on the track.
			//    This value can differ from the initial fStationPosition_X, fStationPosition_Y in case they were not matching the track
			ipTrack[nStationTrackIndex].std.GetMoverPositionAt(fStationPositionOnTrack, StationPosition);
			
			// Providing the station position to e.g. visualization	
			stStationPosition.bInit            := TRUE;
			stStationPosition.fPositionOnTrack := fStationPositionOnTrack;
			stStationPosition.nTrackId         := nStationTrackIndex;
			stStationPosition.fPosition_X	   := StationPosition.x;
			stStationPosition.fPosition_Y	   := StationPosition.y;

			nStateInit := 30;
			
			
	30:		// Clear Lists
			IF THIS^.Clear() THEN
				nStateInit := 90;	
			END_IF

			
		
	90:		// Creating a little history of what happened in the station for debugging purpose
			fbHistoryInfo.AddEntry('Init');
	
			nStateInit := 100;
			
						
	100:	// Init done
			IF SUPER^.Init() THEN
				bStationInitDone := TRUE;	
				           Init := TRUE;
			END_IF
				
	
END_CASE
END_METHOD

METHOD Process : BOOL

VAR_INST
		
	nMoverIndex				: UINT;
	
	fMoverToTrackPosition	: LREAL;
	nTrackIndex				: UINT;
	fMoverVelocity			: LREAL;
	fMoverAcceleration		: LREAL;
	fMoverJerk				: LREAL;
	
	
	nErrorId					: UDINT;
	nObjectID					: UDINT;
	nObjectType					: UDINT;		
	
	// Process
	Timer01						: TON;
	fRotationAngle				: LREAL;
	fRotationVelocity			: LREAL;	
	fRotationAcceleration		: LREAL;
	fRotationJerk				: LREAL;
	stRotationOptions			: ST_MoveCOptions;
	
	nLastMoverDestination		: UINT;
	nNextMoverDestination		: UINT;
	
END_VAR




VAR_INST



//	bToggleSwitch				: BOOL;
//	bStationActive				: BOOL;


//	fPositionOnTrack			: LREAL;
//	nCurrentTrackIndex			: UDINT;
	


//	fInRangePosition			: LREAL;
//	fOutOfRangePosition			: LREAL;
	


	
	
	
//	strInfo						: STRING;
	
					
	

//	ClearTrig					: R_TRIG;
	
//	TrackInfo					: PlanarObjectInfo;
//	nStationTrackID				: UDINT;
//	nMoverOnTrackID				: UDINT;
	

	
//	stMoveOptionsCurve			: ST_MoveCOptions;
//	fVeloTurn           		: LREAL :=   180.0;
//	fAccelTurn    				: LREAL :=  1000.0;
//	fJerkTurn            		: LREAL := 10000.0;	
//	fTurnAngle					: LREAL;	
	

END_VAR
// *** Processing Station ***

CASE nStateProcess OF 

	0:		// Enter
			IF bStationInitDone THEN
				nStateProcess := 100;
			END_IF

	
	100: 	// Waiting for Mover
			IF P_List_Station.P_FirstInList <> 0 THEN
				nMoverIndex := P_List_Station.P_FirstInList.P_Id;
					 nStateProcess := nStateProcess +10;
			END_IF
	
		

	110: 	// Check if Mover is in range
			IF  ipMoverApplication[nMoverIndex].std.P_SetOnTrack.TrackOID = ipTrack[nStationTrackIndex].std.P_OID 
			AND ipMoverApplication[nMoverIndex].std.P_SetOnTrack.SetPos   > fStationPositionOnTrack - fInRangeDistance
			THEN
				nStateProcess := nStateProcess +10;
			END_IF
			
	
	120: 	// Checking process situation
			CASE eProcessMode OF
				
			E_ProcessMode.None:
				;	// Nothing happens -> Process mode needs to be set!
				
			E_ProcessMode.InitRun:
				IF nStationIndex = 1 THEN
					ipMoverApplication[nMoverIndex].P_ProductData.bInitRun := FALSE;
				ELSE
					nStateProcess := 300;
				END_IF				
			
			E_ProcessMode.Production:
				nStateProcess := 200;
		
			END_CASE
		
	
	200: 	// Send mover to Processing-Position
			fMoverToTrackPosition   := fStationPositionOnTrack;
			nTrackIndex        		:= nStationTrackIndex;
			fMoverVelocity     		:=    300.0;
			fMoverAcceleration 		:=  1_000.0;
			fMoverJerk         		:= 10_000.0;	
	
			stMoveParameters.direction := Tc3_Mc3PlanarMotion.MC_DIRECTION.mcDirectionShortestWay;
			stMoveParameters.gap       := 240.0;
		
			
			// Creating info text with a little history of what happened in the station for debugging purpose		
			strInfo := fbHistoryInfo.CreateStationInfo(nStationIndex, nMoverIndex, nNextStationIndex);	


			// Move on track command	
			ipMoverApplication[nMoverIndex].std.MoveOnTrack( strInfo,
															 ipTrack[nTrackIndex].std,
															 fMoverToTrackPosition,
															 fMoverVelocity,
															 fMoverAcceleration,
															 fMoverJerk,
															 stMoveParameters.gap,
															 stMoveParameters.direction);
			nStateProcess := nStateProcess +1;
				
			
	201: 	// Checking move command return
			IF ipMoverApplication[nMoverIndex].std.P_MoveOnTrack.Done THEN
				nStateProcess := nStateProcess +9;
			ELSIF ipMoverApplication[nMoverIndex].std.P_MoveOnTrack.Error THEN
				   nErrorID := ipMoverApplication[nMoverIndex].std.P_MoveOnTrack.ErrorID;
				  nObjectID := ipMoverApplication[nMoverIndex].std.P_MoveOnTrack.stInfo.nObjectID;
				nObjectType := ipMoverApplication[nMoverIndex].std.P_MoveOnTrack.stInfo.nObjectType;
			END_IF		

			
	210:	// Process: Showing mover rotation -> Rotating to +90°
			       fRotationAngle :=   90.0;
			    fRotationVelocity :=  720.0;
			fRotationAcceleration := 1800.0;
			        fRotationJerk := 9000.0;

			stRotationOptions.additionalTurns := 0;
			stRotationOptions.direction		  := Tc3_Mc3PlanarMotion.MC_Direction.mcDirectionNonModulo;

			IF NOT ipMoverApplication[nMoverIndex].std.P_MoveC.Busy THEN
					
				ipMoverApplication[nMoverIndex].std.MoveC( strInfo,
														   fRotationAngle,
														   fRotationVelocity,
														   fRotationAcceleration,
														   fRotationAcceleration,
														   fRotationJerk,
														   stRotationOptions );
														   
				nStateProcess := nStateProcess +1;
			END_IF										   

	211:	// Checking move command return
			IF ipMoverApplication[nMoverIndex].std.P_MoveC.Done THEN
				nStateProcess := nStateProcess +9;
			ELSIF ipMoverApplication[nMoverIndex].std.P_MoveC.Error THEN
				   nErrorID := ipMoverApplication[nMoverIndex].std.P_MoveOnTrack.ErrorID;
				  nObjectID := ipMoverApplication[nMoverIndex].std.P_MoveOnTrack.stInfo.nObjectID;
				nObjectType := ipMoverApplication[nMoverIndex].std.P_MoveOnTrack.stInfo.nObjectType;				
			END_IF			
			
				
	220:	// Process: Rotation-Demo done
			nStateProcess := 300;

		
			
			
	300: 	// Decide to which station the mover needs to travel next.
			nLastMoverDestination := ipMoverApplication[nMoverIndex].P_ProductData.nDestinationProcess;
			CASE nLastMoverDestination OF
			2:	nNextMoverDestination := 3;
			3:	nNextMoverDestination := 2;
			ELSE
				// Mover came in for the first time
				CASE nMoverIndex OF
				1:	nNextMoverDestination := 3;
  				2:	nNextMoverDestination := 2;
				3:	nNextMoverDestination := 2;
  				4:	nNextMoverDestination := 3;				
				END_CASE
			END_CASE
			
			IF  nNextMoverDestination = 2 
			AND ipStation[2].P_ProcessState > 1
			AND ipStation[2].P_ProcessState < 5
			THEN
				nNextMoverDestination := 3;
			END_IF
			
			ipMoverApplication[nMoverIndex].P_ProductData.nDestinationProcess := nNextMoverDestination;
			
			nStateProcess := nStateProcess +10;
		
			
	310:	// Send mover to the next station
			fMoverToTrackPosition   := fSendAwayPosition;	
			nTrackIndex        		:= nStationTrackIndex;		
			fMoverVelocity     		:=    300.0;
			fMoverAcceleration 		:=  1_000.0;
			fMoverJerk         		:= 10_000.0;	
	
			
			stMoveParameters.direction := Tc3_Mc3PlanarMotion.MC_DIRECTION.mcDirectionPositive;	
			stMoveParameters.gap       := 240.0;

			
			// Creating info text with a little history of what happened in the station for debugging purpose		
			strInfo := fbHistoryInfo.CreateStationInfo(nStationIndex, nMoverIndex, nNextStationIndex);	
			
				
			// Move on track command	
			ipMoverApplication[nMoverIndex].std.MoveOnTrack( strInfo,
															 ipTrack[nTrackIndex].std,
															 fMoverToTrackPosition,
															 fMoverVelocity,
															 fMoverAcceleration,
															 fMoverJerk,
															 stMoveParameters.gap,
															 stMoveParameters.direction);
			nStateProcess := nStateProcess +1;
			
		
		
	311: 	// Checking move command return
			IF ipMoverApplication[nMoverIndex].std.P_MoveOnTrack.Active
			OR ipMoverApplication[nMoverIndex].std.P_MoveOnTrack.Done 
			THEN
				nStateProcess := nStateProcess + 9;
				
			ELSIF ipMoverApplication[nMoverIndex].std.P_MoveOnTrack.Error THEN
				   nErrorID := ipMoverApplication[nMoverIndex].std.P_MoveOnTrack.ErrorID;
				  nObjectID := ipMoverApplication[nMoverIndex].std.P_MoveOnTrack.stInfo.nObjectID;
				nObjectType := ipMoverApplication[nMoverIndex].std.P_MoveOnTrack.stInfo.nObjectType;
			END_IF		
		
			
	320: 	// Mover to the list of the next station
			ipStation[nNextStationIndex].P_List_Switch_Input_A.AddMover(P_List_Station.RemoveFirstInList());
			nStateProcess := 500;	
	
		
	500: 	// Done for this cycle
			nStateProcess := 100;

END_CASE
END_METHOD

END_FUNCTION_BLOCK

// ---- 2_Application/Station/Base/FB_StationBase.TcPOU
FUNCTION_BLOCK FB_StationBase IMPLEMENTS I_Station


VAR
	stMoveParameters 	: ST_MoveOnTrackOptions; 	
	stStationPosition	: ST_StationPosition;	
	eProcessMode		: E_ProcessMode;
	StationPosition     : PositionXYC;	
	
	idx  				: UDINT;
	nStateInit			: UDINT;
	nStateClear 		: UDINT;
	nStateProcess		: UDINT;
	bStationInitDone	: BOOL;	
	
	
	// Lists for Stations
	fbList_Station		: FB_List;
	fbList_InputA		: FB_List;		
	fbList_InputB		: FB_List;	
	fbList_InputC		: FB_List;		

	
	// History info for debugging purpose
	strInfo				: STRING;	
	fbHistoryInfo		: FB_HistoryInfo;	
	
	
	nProcessRequest		: DINT;
	nProcessClearence	: DINT;
	nProcessState		: DINT;
	
	fStationPositionOnTrack		: LREAL;	
END_VAR

METHOD Clear : BOOL
VAR_INPUT
END_VAR


VAR_INST

	nStateClear : UINT;

END_VAR


	CASE nStateClear OF 
		
	0:	// Enter
		            Clear := FALSE;
		  nProcessRequest := 0;
		nProcessClearence := 0;
		    nProcessState := 0;	  
			  
		nStateClear := nStateClear +10;
		
	10: // Clear Station-List
		IF fbList_Station.ClearList() THEN
			nStateClear := nStateClear +10;	
		END_IF
		
	20: // Clear InputA-List
		IF fbList_InputA.ClearList() THEN
			nStateClear := nStateClear +10;	
		END_IF
	
	30: // Clear InputB-List
		IF fbList_InputB.ClearList() THEN
			nStateClear := nStateClear +10;	
		END_IF	
	
	40: // Clear InputC-List
		IF fbList_InputB.ClearList() THEN
			nStateClear := nStateClear +10;	
		END_IF		
	
	50:	nStateClear := 100;	
		
		
	100:  // Done
		nStateClear := 0;
		      Clear := TRUE;
		
	END_CASE
END_METHOD

METHOD Cycle : BOOL
VAR_INPUT
END_VAR
VAR
	nForCounter : INT;
END_VAR


VAR_INST
	
	fTestValueX	: LREAL;
	fTestValueY : LREAL;	
	
END_VAR
;
END_METHOD

METHOD Init : BOOL


	  nStateInit := 0;
	nStateProcess := 0;
	 eProcessMode := E_ProcessMode.None;

	Init := TRUE;
END_METHOD

PROPERTY P_bInitDone : BOOL
GET
P_bInitDone := bStationInitDone;
END_GET
END_PROPERTY

PROPERTY P_eProcessMode : E_ProcessMode
GET
P_eProcessMode := eProcessMode;
END_GET
SET
eProcessMode := P_eProcessMode;
END_SET
END_PROPERTY

PROPERTY P_List_Station : I_List
GET
P_List_Station := fbList_Station;
END_GET
END_PROPERTY

PROPERTY P_List_Switch_Input_A : I_List
GET
P_List_Switch_Input_A := fbList_InputA;
END_GET
END_PROPERTY

PROPERTY P_List_Switch_Input_B : I_List
GET
P_List_Switch_Input_B := fbList_InputB;
END_GET
END_PROPERTY

PROPERTY P_List_Switch_Input_C : I_List
GET
P_List_Switch_Input_C := fbList_InputC;
END_GET
END_PROPERTY

PROPERTY P_nErrorCode : UDINT
GET
END_GET
END_PROPERTY

PROPERTY P_Position : ST_StationPosition
GET
P_Position := stStationPosition;
END_GET
END_PROPERTY

PROPERTY P_ProcessClearance : DINT
GET
P_ProcessClearance := nProcessClearence;
END_GET
END_PROPERTY

PROPERTY P_ProcessRequest : DINT
GET
P_ProcessRequest := nProcessRequest;
END_GET
SET
nProcessRequest := P_ProcessRequest;
END_SET
END_PROPERTY

PROPERTY P_ProcessState : DINT
GET
P_ProcessState := nProcessState;
END_GET
END_PROPERTY

METHOD Process : BOOL
;
END_METHOD

END_FUNCTION_BLOCK

// ---- 2_Application/Station/Helper/FB_HistoryInfo.TcPOU
FUNCTION_BLOCK FB_HistoryInfo


VAR
	strInfo				: STRING;
	strInfoHistory		: ARRAY[0..10] OF STRING;
END_VAR

METHOD AddEntry : BOOL
VAR_INPUT
	sInfo	: STRING;
END_VAR


VAR
	idx	: UDINT;
END_VAR


	FOR idx:=10 TO 1 BY -1 DO 
		strInfoHistory[idx] := strInfoHistory[idx-1];
	END_FOR
	strInfoHistory[0] := sInfo;
END_METHOD

METHOD CreateStationInfo : STRING
VAR_INPUT
	nStationIndex		: UDINT;
	nMoverIndex			: UDINT;
	nNextStationIndex   : UDINT;
END_VAR



VAR
	strInfo			: STRING;	
END_VAR


	strInfo := CONCAT('St:', UDINT_TO_STRING(nStationIndex));
	strInfo := CONCAT(strInfo, ' M:');
	strInfo := CONCAT(strInfo, UDINT_TO_STRING(nMoverIndex));
	strInfo := CONCAT(strInfo, ' to next station:');
	strInfo := CONCAT(strInfo, UDINT_TO_STRING(nNextStationIndex));
	
	CreateStationInfo := strInfo;		
			
	THIS^.AddEntry(strInfo);
END_METHOD

END_FUNCTION_BLOCK

// ---- 2_Application/Station/FB_Station_02_Process.TcPOU
FUNCTION_BLOCK FB_Station_02_Process EXTENDS FB_StationBase
VAR
	nStationIndex				: UINT;
	nNextStationIndex			: UINT;
	nStationTrackIndex			: UINT;
	
	fStationPosition_X 			: LREAL;
	fStationPosition_Y 			: LREAL;		  
    fSendAwayDistance			: LREAL;	
	fInRangeDistance			: LREAL;	
	fSendAwayPosition			: LREAL;
	
	position					: PositionXYC;

END_VAR

METHOD Clear : BOOL
VAR_INPUT
END_VAR



	CASE nStateClear OF
		
	0:	// Enter
		Clear := FALSE;
		nStateClear := nStateClear +10;
		
	10: // Clearing all Station-Lists 
		IF SUPER^.Clear() THEN
			nStateClear := nStateClear +10;
		END_IF	
	
	20:	// Add aditional Data to be cleared here...
		nStateClear := 100;
		
		
	100: // Done
		      Clear := TRUE;
		nStateClear := 0;

	END_CASE
END_METHOD

METHOD Init : BOOL



VAR_INST
	nTestCounter	: INT;	
END_VAR
nTestCounter := nTestCounter +1;

CASE nStateInit OF

	0:		// Enter 
			bStationInitDone := FALSE;
			   nStateProcess := 0;
			      nStateInit := 10;
				 
			
	10:		// Init Station-Parameters				
				  nStationIndex := 2;				// Each station needs an unique index	
			 nStationTrackIndex := 2;	 			// Track on which the station resides
			  nNextStationIndex := 5;				// Index of the following station 
							  
			 fStationPosition_X := 600.0;			// Position of the station in X/Y coordinates
			 fStationPosition_Y := 360.0;			// Position of the station in X/Y coordinates
			  
			  fSendAwayDistance :=   5.0;			// Position on track a mover will be send to after processing 
			  fInRangeDistance  := 300.0;			// Position in front of a station from where a mover will be taken over
			  
			  nStateInit := 11;
				   
				  
	11: // Fail-safe check, just to make sure all variables have been assigned after doing copy&paste from the template
			IF        nStationIndex > 0
			AND  nStationTrackIndex > 0
			AND   nNextStationIndex > 0
			AND  fStationPosition_X > 0
			AND  fStationPosition_Y > 0
			AND   fSendAwayDistance > 0
			THEN   
				nStateInit := 20;
			END_IF
			
				   
	20:		// Calculating positions
	
			// 1. Calculating station position on track
			position.SetValuesXYC(fStationPosition_X, fStationPosition_Y, 0.0);
			fStationPositionOnTrack := ipTrack[nStationTrackIndex].std.GetTrackPositionAt(position);
							
			// 2. Calculating send-away position on track
			fSendAwayPosition := fStationPositionOnTrack + fSendAwayDistance; 
			
			// The send away position must not exceed the lenght of the track!
			IF fSendAwayPosition > ipTrack[nStationTrackIndex].P_TrackLength THEN
				fSendAwayPosition := ipTrack[nStationTrackIndex].P_TrackLength;
			END_IF
			
			// 3. Calculating the station position in X/Y coordinates determined by the track	
            //    This is to make sure the center of the station is always located directly on the track.
			//    This value can differ from the initial fStationPosition_X, fStationPosition_Y in case they were not matching the track
			ipTrack[nStationTrackIndex].std.GetMoverPositionAt(fStationPositionOnTrack, StationPosition);
			
			// Providing the station position to e.g. visualization	
			stStationPosition.bInit            := TRUE;
			stStationPosition.fPositionOnTrack := fStationPositionOnTrack;
			stStationPosition.nTrackId         := nStationTrackIndex;
			stStationPosition.fPosition_X	   := StationPosition.x;
			stStationPosition.fPosition_Y	   := StationPosition.y;

			nStateInit := 30;
			
			
	30:		// Clear Lists
			IF THIS^.Clear() THEN
				nStateInit := 90;	
			END_IF

			

	90:		// Creating a little history of what happened in the station for debugging purpose
			fbHistoryInfo.AddEntry('Init');
	
			nStateInit := 100;
			
						
	100:	// Init done
			IF SUPER^.Init() THEN
				bStationInitDone := TRUE;	
				           Init := TRUE;
			END_IF
				
	
END_CASE
END_METHOD

METHOD Process : BOOL

VAR_INST
		
	nMoverIndex				: UINT;
	
	fMoverToTrackPosition	: LREAL;
	nTrackIndex				: UINT;
	fMoverVelocity			: LREAL;
	fMoverAcceleration		: LREAL;
	fMoverJerk				: LREAL;
	
	
	nErrorId					: UDINT;
	nObjectID					: UDINT;
	nObjectType					: UDINT;		
	
	// Process
	Timer01						: TON;
	fRotationAngle				: LREAL;
	fRotationVelocity			: LREAL;	
	fRotationAcceleration		: LREAL;
	fRotationJerk				: LREAL;
	stRotationOptions			: ST_MoveCOptions;
	
	
	
	
END_VAR




VAR_INST



//	bToggleSwitch				: BOOL;
//	bStationActive				: BOOL;


//	fPositionOnTrack			: LREAL;
//	nCurrentTrackIndex			: UDINT;
	


//	fInRangePosition			: LREAL;
//	fOutOfRangePosition			: LREAL;
	


	
	
	
//	strInfo						: STRING;
	
					
	

//	ClearTrig					: R_TRIG;
	
//	TrackInfo					: PlanarObjectInfo;
//	nStationTrackID				: UDINT;
//	nMoverOnTrackID				: UDINT;
	

	
//	stMoveOptionsCurve			: ST_MoveCOptions;
//	fVeloTurn           		: LREAL :=   180.0;
//	fAccelTurn    				: LREAL :=  1000.0;
//	fJerkTurn            		: LREAL := 10000.0;	
//	fTurnAngle					: LREAL;	
	

END_VAR


// *** Processing Station ***

CASE nStateProcess OF 

	0:		// Enter
			IF bStationInitDone THEN
				nStateProcess := 100;
			END_IF

	
	100: 	// Waiting for Mover
			IF P_List_Station.P_FirstInList <> 0 THEN
				nMoverIndex := P_List_Station.P_FirstInList.P_Id;
					 nStateProcess := nStateProcess +10;
			END_IF
	
		
	110: 	// Check if Mover is in range
			IF  ipMoverApplication[nMoverIndex].std.P_SetOnTrack.TrackOID = ipTrack[nStationTrackIndex].std.P_OID 
			AND ipMoverApplication[nMoverIndex].std.P_SetOnTrack.SetPos   > fStationPositionOnTrack - fInRangeDistance
			THEN
				nStateProcess := nStateProcess +10;
			END_IF
			
	
	120: 	// Checking process situation
			CASE eProcessMode OF
				
			E_ProcessMode.None:
				;	// Nothing happens -> Process mode needs to be set!
				
			E_ProcessMode.InitRun:
				IF nStationIndex = 1 THEN
					ipMoverApplication[nMoverIndex].P_ProductData.bInitRun := FALSE;
				ELSE
					nStateProcess := 300;
				END_IF				
			
			E_ProcessMode.Production:
				nStateProcess := 200;
		
			END_CASE
		
	
	200: 	// Send mover to Processing-Position
			fMoverToTrackPosition   := fStationPositionOnTrack;
			nTrackIndex        		:= nStationTrackIndex;
			fMoverVelocity     		:=    300.0;
			fMoverAcceleration 		:=  1_000.0;
			fMoverJerk         		:= 10_000.0;	
	
			stMoveParameters.direction := Tc3_Mc3PlanarMotion.MC_DIRECTION.mcDirectionShortestWay;
			stMoveParameters.gap       := 240.0;
		
			
			// Creating info text with a little history of what happened in the station for debugging purpose		
			strInfo := fbHistoryInfo.CreateStationInfo(nStationIndex, nMoverIndex, nNextStationIndex);	


			// Move on track command	
			ipMoverApplication[nMoverIndex].std.MoveOnTrack( strInfo,
															 ipTrack[nTrackIndex].std,
															 fMoverToTrackPosition,
															 fMoverVelocity,
															 fMoverAcceleration,
															 fMoverJerk,
															 stMoveParameters.gap,
															 stMoveParameters.direction);
			nStateProcess := nStateProcess +1;
				
			
	201: 	// Checking move command return
			IF ipMoverApplication[nMoverIndex].std.P_MoveOnTrack.Done THEN
				nStateProcess := nStateProcess +9;
			ELSIF ipMoverApplication[nMoverIndex].std.P_MoveOnTrack.Error THEN
				   nErrorID := ipMoverApplication[nMoverIndex].std.P_MoveOnTrack.ErrorID;
				  nObjectID := ipMoverApplication[nMoverIndex].std.P_MoveOnTrack.stInfo.nObjectID;
				nObjectType := ipMoverApplication[nMoverIndex].std.P_MoveOnTrack.stInfo.nObjectType;
			END_IF		

			
	210:	// Process: Showing mover rotation -> Rotating 180°
			       fRotationAngle :=  360.0;
			    fRotationVelocity :=  180.0;
			fRotationAcceleration := 1800.0;
			        fRotationJerk := 9000.0;

